DATA_BLOCK "DB_DigIn_I3.6"   // DB138
{ S7_Optimized_Access := 'TRUE' }
VERSION : 0.1
// stored: InstanceOfName FB_DigIn
"FB_DigIn"
BEGIN
END_DATA_BLOCK

DATA_BLOCK "DB_DigIn_I3.7"   // DB139
{ S7_Optimized_Access := 'TRUE' }
VERSION : 0.1
// stored: InstanceOfName FB_DigIn
"FB_DigIn"
BEGIN
END_DATA_BLOCK

DATA_BLOCK "DB_DigIn_I4.0"   // DB140
{ S7_Optimized_Access := 'TRUE' }
VERSION : 0.1
// stored: InstanceOfName FB_DigIn
"FB_DigIn"
BEGIN
END_DATA_BLOCK

DATA_BLOCK "DB_DigIn_I4.1"   // DB141
{ S7_Optimized_Access := 'TRUE' }
VERSION : 0.1
// stored: InstanceOfName FB_DigIn
"FB_DigIn"
BEGIN
END_DATA_BLOCK

DATA_BLOCK "DB_DigIn_I4.2"   // DB142
{ S7_Optimized_Access := 'TRUE' }
VERSION : 0.1
// stored: InstanceOfName FB_DigIn
"FB_DigIn"
BEGIN
END_DATA_BLOCK

DATA_BLOCK "DB_DigIn_I4.3"   // DB143
{ S7_Optimized_Access := 'TRUE' }
VERSION : 0.1
// stored: InstanceOfName FB_DigIn
"FB_DigIn"
BEGIN
END_DATA_BLOCK

DATA_BLOCK "DB_DigIn_I4.4"   // DB144
{ S7_Optimized_Access := 'TRUE' }
VERSION : 0.1
// stored: InstanceOfName FB_DigIn
"FB_DigIn"
BEGIN
END_DATA_BLOCK

DATA_BLOCK "DB_DigIn_I4.5"   // DB145
{ S7_Optimized_Access := 'TRUE' }
VERSION : 0.1
// stored: InstanceOfName FB_DigIn
"FB_DigIn"
BEGIN
END_DATA_BLOCK

DATA_BLOCK "DB_DigIn_I4.6"   // DB146
{ S7_Optimized_Access := 'TRUE' }
VERSION : 0.1
// stored: InstanceOfName FB_DigIn
"FB_DigIn"
BEGIN
END_DATA_BLOCK

DATA_BLOCK "DB_DigIn_I4.7"   // DB147
{ S7_Optimized_Access := 'TRUE' }
VERSION : 0.1
// stored: InstanceOfName FB_DigIn
"FB_DigIn"
BEGIN
END_DATA_BLOCK

DATA_BLOCK "DB_DigIn_I5.0"   // DB148
{ S7_Optimized_Access := 'TRUE' }
VERSION : 0.1
// stored: InstanceOfName FB_DigIn
"FB_DigIn"
BEGIN
END_DATA_BLOCK

DATA_BLOCK "DB_DigIn_I5.1"   // DB149
{ S7_Optimized_Access := 'TRUE' }
VERSION : 0.1
// stored: InstanceOfName FB_DigIn
"FB_DigIn"
BEGIN
END_DATA_BLOCK

DATA_BLOCK "DB_DigIn_I5.2"   // DB150
{ S7_Optimized_Access := 'TRUE' }
VERSION : 0.1
// stored: InstanceOfName FB_DigIn
"FB_DigIn"
BEGIN
END_DATA_BLOCK

DATA_BLOCK "DB_DigIn_I5.3"   // DB151
{ S7_Optimized_Access := 'TRUE' }
VERSION : 0.1
// stored: InstanceOfName FB_DigIn
"FB_DigIn"
BEGIN
END_DATA_BLOCK

DATA_BLOCK "DB_DigIn_I5.4"   // DB152
{ S7_Optimized_Access := 'TRUE' }
VERSION : 0.1
// stored: InstanceOfName FB_DigIn
"FB_DigIn"
BEGIN
END_DATA_BLOCK

DATA_BLOCK "DB_DigIn_I5.5"   // DB153
{ S7_Optimized_Access := 'TRUE' }
VERSION : 0.1
// stored: InstanceOfName FB_DigIn
"FB_DigIn"
BEGIN
END_DATA_BLOCK

DATA_BLOCK "DB_DigIn_I5.6"   // DB154
{ S7_Optimized_Access := 'TRUE' }
VERSION : 0.1
// stored: InstanceOfName FB_DigIn
"FB_DigIn"
BEGIN
END_DATA_BLOCK

DATA_BLOCK "DB_DigIn_I5.7"   // DB155
{ S7_Optimized_Access := 'TRUE' }
VERSION : 0.1
// stored: InstanceOfName FB_DigIn
"FB_DigIn"
BEGIN
END_DATA_BLOCK

DATA_BLOCK "DB_DigIn_I6.0"   // DB156
{ S7_Optimized_Access := 'TRUE' }
VERSION : 0.1
// stored: InstanceOfName FB_DigIn
"FB_DigIn"
BEGIN
END_DATA_BLOCK

DATA_BLOCK "DB_DigIn_I6.1"   // DB157
{ S7_Optimized_Access := 'TRUE' }
VERSION : 0.1
// stored: InstanceOfName FB_DigIn
"FB_DigIn"
BEGIN
END_DATA_BLOCK

DATA_BLOCK "DB_DigIn_I6.2"   // DB158
{ S7_Optimized_Access := 'TRUE' }
VERSION : 0.1
// stored: InstanceOfName FB_DigIn
"FB_DigIn"
BEGIN
END_DATA_BLOCK

DATA_BLOCK "DB_DigIn_I6.3"   // DB159
{ S7_Optimized_Access := 'TRUE' }
VERSION : 0.1
// stored: InstanceOfName FB_DigIn
"FB_DigIn"
BEGIN
END_DATA_BLOCK

DATA_BLOCK "DB_DigIn_I6.4"   // DB160
{ S7_Optimized_Access := 'TRUE' }
VERSION : 0.1
// stored: InstanceOfName FB_DigIn
"FB_DigIn"
BEGIN
END_DATA_BLOCK

DATA_BLOCK "DB_DigIn_I6.5"   // DB161
{ S7_Optimized_Access := 'TRUE' }
VERSION : 0.1
// stored: InstanceOfName FB_DigIn
"FB_DigIn"
BEGIN
END_DATA_BLOCK

DATA_BLOCK "DB_DigIn_I6.6"   // DB162
{ S7_Optimized_Access := 'TRUE' }
VERSION : 0.1
// stored: InstanceOfName FB_DigIn
"FB_DigIn"
BEGIN
END_DATA_BLOCK

DATA_BLOCK "DB_DigIn_I6.7"   // DB163
{ S7_Optimized_Access := 'TRUE' }
VERSION : 0.1
// stored: InstanceOfName FB_DigIn
"FB_DigIn"
BEGIN
END_DATA_BLOCK

DATA_BLOCK "DB_DigIn_I7.0"   // DB164
{ S7_Optimized_Access := 'TRUE' }
VERSION : 0.1
// stored: InstanceOfName FB_DigIn
"FB_DigIn"
BEGIN
END_DATA_BLOCK

DATA_BLOCK "DB_DigIn_I7.1"   // DB165
{ S7_Optimized_Access := 'TRUE' }
VERSION : 0.1
// stored: InstanceOfName FB_DigIn
"FB_DigIn"
BEGIN
END_DATA_BLOCK

DATA_BLOCK "DB_DigIn_I7.2"   // DB166
{ S7_Optimized_Access := 'TRUE' }
VERSION : 0.1
// stored: InstanceOfName FB_DigIn
"FB_DigIn"
BEGIN
END_DATA_BLOCK

DATA_BLOCK "DB_DigIn_I7.3"   // DB167
{ S7_Optimized_Access := 'TRUE' }
VERSION : 0.1
// stored: InstanceOfName FB_DigIn
"FB_DigIn"
BEGIN
END_DATA_BLOCK

DATA_BLOCK "DB_DigIn_I7.4"   // DB168
{ S7_Optimized_Access := 'TRUE' }
VERSION : 0.1
// stored: InstanceOfName FB_DigIn
"FB_DigIn"
BEGIN
END_DATA_BLOCK

DATA_BLOCK "DB_DigIn_I7.5"   // DB169
{ S7_Optimized_Access := 'TRUE' }
VERSION : 0.1
// stored: InstanceOfName FB_DigIn
"FB_DigIn"
BEGIN
END_DATA_BLOCK

DATA_BLOCK "DB_DigIn_I7.6"   // DB170
{ S7_Optimized_Access := 'TRUE' }
VERSION : 0.1
// stored: InstanceOfName FB_DigIn
"FB_DigIn"
BEGIN
END_DATA_BLOCK

DATA_BLOCK "DB_DigIn_I7.7"   // DB171
{ S7_Optimized_Access := 'TRUE' }
VERSION : 0.1
// stored: InstanceOfName FB_DigIn
"FB_DigIn"
BEGIN
END_DATA_BLOCK

DATA_BLOCK "DB_DigOut_Q0.0"   // DB172
{ S7_Optimized_Access := 'TRUE' }
VERSION : 0.1
// stored: InstanceOfName FB_DigOut
"FB_DigOut"
BEGIN
END_DATA_BLOCK

DATA_BLOCK "DB_DigOut_Q0.1"   // DB173
{ S7_Optimized_Access := 'TRUE' }
VERSION : 0.1
// stored: InstanceOfName FB_DigOut
"FB_DigOut"
BEGIN
END_DATA_BLOCK

DATA_BLOCK "DB_DigOut_Q0.2"   // DB174
{ S7_Optimized_Access := 'TRUE' }
VERSION : 0.1
// stored: InstanceOfName FB_DigOut
"FB_DigOut"
BEGIN
END_DATA_BLOCK

DATA_BLOCK "DB_DigOut_Q0.3"   // DB175
{ S7_Optimized_Access := 'TRUE' }
VERSION : 0.1
// stored: InstanceOfName FB_DigOut
"FB_DigOut"
BEGIN
END_DATA_BLOCK

DATA_BLOCK "DB_DigOut_Q0.4"   // DB176
{ S7_Optimized_Access := 'TRUE' }
VERSION : 0.1
// stored: InstanceOfName FB_DigOut
"FB_DigOut"
BEGIN
END_DATA_BLOCK

DATA_BLOCK "DB_DigOut_Q0.5"   // DB177
{ S7_Optimized_Access := 'TRUE' }
VERSION : 0.1
// stored: InstanceOfName FB_DigOut
"FB_DigOut"
BEGIN
END_DATA_BLOCK

DATA_BLOCK "DB_DigOut_Q0.6"   // DB178
{ S7_Optimized_Access := 'TRUE' }
VERSION : 0.1
// stored: InstanceOfName FB_DigOut
"FB_DigOut"
BEGIN
END_DATA_BLOCK

DATA_BLOCK "DB_DigOut_Q0.7"   // DB179
{ S7_Optimized_Access := 'TRUE' }
VERSION : 0.1
// stored: InstanceOfName FB_DigOut
"FB_DigOut"
BEGIN
END_DATA_BLOCK

DATA_BLOCK "DB_DigOut_Q1.0"   // DB180
{ S7_Optimized_Access := 'TRUE' }
VERSION : 0.1
// stored: InstanceOfName FB_DigOut
"FB_DigOut"
BEGIN
END_DATA_BLOCK

DATA_BLOCK "DB_DigOut_Q1.1"   // DB181
{ S7_Optimized_Access := 'TRUE' }
VERSION : 0.1
// stored: InstanceOfName FB_DigOut
"FB_DigOut"
BEGIN
END_DATA_BLOCK

DATA_BLOCK "DB_DigOut_Q1.2"   // DB182
{ S7_Optimized_Access := 'TRUE' }
VERSION : 0.1
// stored: InstanceOfName FB_DigOut
"FB_DigOut"
BEGIN
END_DATA_BLOCK

DATA_BLOCK "DB_DigOut_Q1.3"   // DB183
{ S7_Optimized_Access := 'TRUE' }
VERSION : 0.1
// stored: InstanceOfName FB_DigOut
"FB_DigOut"
BEGIN
END_DATA_BLOCK

DATA_BLOCK "DB_DigOut_Q1.4"   // DB184
{ S7_Optimized_Access := 'TRUE' }
VERSION : 0.1
// stored: InstanceOfName FB_DigOut
"FB_DigOut"
BEGIN
END_DATA_BLOCK

DATA_BLOCK "DB_DigOut_Q1.5"   // DB185
{ S7_Optimized_Access := 'TRUE' }
VERSION : 0.1
// stored: InstanceOfName FB_DigOut
"FB_DigOut"
BEGIN
END_DATA_BLOCK

DATA_BLOCK "DB_DigOut_Q1.6"   // DB186
{ S7_Optimized_Access := 'TRUE' }
VERSION : 0.1
// stored: InstanceOfName FB_DigOut
"FB_DigOut"
BEGIN
END_DATA_BLOCK

DATA_BLOCK "DB_DigOut_Q1.7"   // DB187
{ S7_Optimized_Access := 'TRUE' }
VERSION : 0.1
// stored: InstanceOfName FB_DigOut
"FB_DigOut"
BEGIN
END_DATA_BLOCK

// folder: 2000_Tools

DATA_BLOCK "FB_Bell_DB"   // DB2003
{ S7_Optimized_Access := 'TRUE' }
VERSION : 0.1
// stored: InstanceOfName FB_Bell
"FB_Bell"
BEGIN
END_DATA_BLOCK

// folder: 20_PSM/PSM_DB

DATA_BLOCK "DB_PSM_LC"   // DB20
{ S7_Optimized_Access := 'TRUE' }
VERSION : 0.1
// stored: InstanceOfName FB_PSM_LC
"FB_PSM_LC"
BEGIN
END_DATA_BLOCK

DATA_BLOCK "DB_PSM_Messages"   // DB21
{ S7_Optimized_Access := 'TRUE' }
VERSION : 0.1
// stored: InstanceOfName FB_PSM_Messages
"FB_PSM_Messages"
BEGIN
END_DATA_BLOCK

DATA_BLOCK "DB_PSM_Alarms"   // DB22
{ S7_Optimized_Access := 'TRUE' }
VERSION : 0.1
// stored: InstanceOfName FB_PSM_Alarms
"FB_PSM_Alarms"
BEGIN
END_DATA_BLOCK

// folder: 300_1UZ1_Lifting(LM)/LM_DB

DATA_BLOCK "DB_Lifting_Control"   // DB300
{ S7_Optimized_Access := 'TRUE' }
VERSION : 0.1
// stored: InstanceOfName FB_Lifting_Control
"FB_Lifting_Control"
BEGIN
END_DATA_BLOCK

DATA_BLOCK "DB_LiftUp_Messages"   // DB321
{ S7_Optimized_Access := 'TRUE' }
VERSION : 0.1
// stored: InstanceOfName FB_LiftUp_Messages
"FB_LiftUp_Messages"
BEGIN
END_DATA_BLOCK

// folder: 400_3UZ1_Trolley_movement(TM)/TM_DB

DATA_BLOCK "DB_Trolley_Control"   // DB400
{ S7_Optimized_Access := 'TRUE' }
VERSION : 0.1
// stored: InstanceOfName FB_Trolley_Control
"FB_Trolley_Control"
BEGIN
END_DATA_BLOCK

DATA_BLOCK "DB_Trolley_Messages"   // DB421
{ S7_Optimized_Access := 'TRUE' }
VERSION : 0.1
// stored: InstanceOfName FB_Trolley_Messages
"FB_Trolley_Messages"
BEGIN
END_DATA_BLOCK

// folder: 500_4UZ1_4UZ2_Crane_movement(CM)/CM_DB

DATA_BLOCK "DB_Crane_Control"   // DB500
{ S7_Optimized_Access := 'TRUE' }
VERSION : 0.1
// stored: InstanceOfName FB_Crane_Control
"FB_Crane_Control"
BEGIN
END_DATA_BLOCK

DATA_BLOCK "DB_Crane_Messages"   // DB521
{ S7_Optimized_Access := 'TRUE' }
VERSION : 0.1
// stored: InstanceOfName FB_Crane_Messages
"FB_Crane_Messages"
BEGIN
END_DATA_BLOCK

// folder: 50_Drives/Drives_DB

DATA_BLOCK "DB_CU_U1"   // DB50
{ S7_Optimized_Access := 'TRUE' }
VERSION : 0.1
// stored: InstanceOfName FB_S120_Tel390_CU
"FB_S120_Tel390_CU"
BEGIN
END_DATA_BLOCK

DATA_BLOCK "DB_Drive_1UZ1"   // DB51
{ S7_Optimized_Access := 'TRUE' }
VERSION : 0.1
// stored: InstanceOfName FB_S120_Tel220
"FB_S120_Tel220"
BEGIN
END_DATA_BLOCK

DATA_BLOCK "DB_Drive_3UZ1"   // DB52
{ S7_Optimized_Access := 'TRUE' }
VERSION : 0.1
// stored: InstanceOfName FB_S120_Tel220
"FB_S120_Tel220"
BEGIN
END_DATA_BLOCK

DATA_BLOCK "DB_Drive_4UZ1"   // DB53
{ S7_Optimized_Access := 'TRUE' }
VERSION : 0.1
// stored: InstanceOfName FB_S120_Tel220
"FB_S120_Tel220"
BEGIN
END_DATA_BLOCK

DATA_BLOCK "DB_Drive_4UZ2"   // DB54
{ S7_Optimized_Access := 'TRUE' }
VERSION : 0.1
// stored: InstanceOfName FB_S120_Tel220
"FB_S120_Tel220"
BEGIN
END_DATA_BLOCK

DATA_BLOCK "DB_Drives_Test"   // DB55
{ S7_Optimized_Access := 'TRUE' }
VERSION : 0.1
   VAR
      Sim_On : Bool := False;
      Sim_Reset : Bool := False;
      U1 : Struct   // Блок керування CU320-2PN
         Enable : Bool := True;
         Ack : Bool := False;
      END_STRUCT;
      "1UZ1" : Struct   // Привід підйому
         Enable : Bool := False;
         Ack : Bool := False;
         SpeedSp : Real := 0.0;
         QuickStop : Bool := False;
         CoastStop : Bool := False;
         SimFault : Bool := False;
         SimWarning : Bool := False;
      END_STRUCT;
      "3UZ1" : Struct   // Привод візка
         Enable : Bool := False;
         Ack : Bool := False;
         SpeedSp : Real := 0.0;
         QuickStop : Bool := False;
         CoastStop : Bool := False;
         SimFault : Bool := False;
         SimWarning : Bool := False;
      END_STRUCT;
      "4UZ1" : Struct   // Привод моста 1
         Enable : Bool := False;
         Ack : Bool := False;
         SpeedSp : Real := 0.0;
         QuickStop : Bool := False;
         CoastStop : Bool := False;
         SimFault : Bool := False;
         SimWarning : Bool := False;
      END_STRUCT;
      "4UZ2" : Struct   // Привод моста 2
         Enable : Bool := False;
         Ack : Bool := False;
         SpeedSp : Real := 0.0;
         QuickStop : Bool := False;
         CoastStop : Bool := False;
         SimFault : Bool := False;
         SimWarning : Bool := False;
      END_STRUCT;
   END_VAR
BEGIN
END_DATA_BLOCK

// folder: 600_Diagnostic

DATA_BLOCK "FB_DIAG_SCALANCE_NODE_DB"   // DB609
{ S7_Optimized_Access := 'TRUE' }
AUTHOR : PIA
FAMILY : System
VERSION : 0.1
// stored: InstanceOfName FB_DIAG_NODE
"FB_DIAG_NODE"
BEGIN
END_DATA_BLOCK

DATA_BLOCK "DB_HMI_Connection"   // DB631
{ S7_Optimized_Access := 'FALSE' }
VERSION : 0.1
// DB631. Постійна ознака доступності даних ПЛК для HMI. Не потребує виклику в OB1. Опитування RUN/STOP використовує існуючу область HMI_DB.wCoordination.
   VAR
      Available : Bool := true;   // Постійне TRUE для перевірки звʼязку з HMI. Після помилки звʼязку панель локально підставляє FALSE; значення у DB не змінюється.
   END_VAR
BEGIN
END_DATA_BLOCK

// folder: 600_Diagnostic/Diag_DB

DATA_BLOCK "DB_SCALANCE"   // DB600
{ S7_Optimized_Access := 'TRUE' }
AUTHOR : PIA
FAMILY : System
VERSION : 0.1
// stored: InstanceOfName FB_DIAG_SCALANCE
"FB_DIAG_SCALANCE"
BEGIN
END_DATA_BLOCK

DATA_BLOCK "DB_DIAG_NODE"   // DB601
{ S7_Optimized_Access := 'TRUE' }
AUTHOR : PIA
FAMILY : System
VERSION : 0.1
// stored: InstanceOfName FB_DIAG_NODE
"FB_DIAG_NODE"
BEGIN
END_DATA_BLOCK

DATA_BLOCK "DB_DIAG_ENC_1BR_NODE"   // DB602
{ S7_Optimized_Access := 'TRUE' }
AUTHOR : PIA
FAMILY : System
VERSION : 0.1
// stored: InstanceOfName FB_DIAG_NODE
"FB_DIAG_NODE"
BEGIN
END_DATA_BLOCK

DATA_BLOCK "DB_DIAG_ENC_3BR_NODE"   // DB603
{ S7_Optimized_Access := 'TRUE' }
AUTHOR : PIA
FAMILY : System
VERSION : 0.1
// stored: InstanceOfName FB_DIAG_NODE
"FB_DIAG_NODE"
BEGIN
END_DATA_BLOCK

DATA_BLOCK "DB_DIAG_ENC_4BR1_NODE"   // DB604
{ S7_Optimized_Access := 'TRUE' }
AUTHOR : PIA
FAMILY : System
VERSION : 0.1
// stored: InstanceOfName FB_DIAG_NODE
"FB_DIAG_NODE"
BEGIN
END_DATA_BLOCK

DATA_BLOCK "DB_DIAG_ENC_4BR2_NODE"   // DB605
{ S7_Optimized_Access := 'TRUE' }
AUTHOR : PIA
FAMILY : System
VERSION : 0.1
// stored: InstanceOfName FB_DIAG_NODE
"FB_DIAG_NODE"
BEGIN
END_DATA_BLOCK

DATA_BLOCK "DB_DIAG_CU320_NODE"   // DB606
{ S7_Optimized_Access := 'TRUE' }
AUTHOR : PIA
FAMILY : System
VERSION : 0.1
// stored: InstanceOfName FB_DIAG_NODE
"FB_DIAG_NODE"
BEGIN
END_DATA_BLOCK

DATA_BLOCK "DB_DIAG_SCALANCE"   // DB607
{ S7_Optimized_Access := 'TRUE' }
AUTHOR : PIA
FAMILY : System
VERSION : 0.1
// stored: InstanceOfName FB_DIAG_SCALANCE
"FB_DIAG_SCALANCE"
BEGIN
END_DATA_BLOCK

DATA_BLOCK "DB_Diagnostics_Messages"   // DB621
{ S7_Optimized_Access := 'TRUE' }
VERSION : 0.1
// stored: InstanceOfName FB_Diagnostics_Messages
"FB_Diagnostics_Messages"
BEGIN
END_DATA_BLOCK

DATA_BLOCK "DB_Diag_Prof"   // DB630
{ S7_Optimized_Access := 'TRUE' }
VERSION : 0.1
// stored: InstanceOfName FB_Diag_MRP
"FB_Diag_MRP"
BEGIN
END_DATA_BLOCK

// folder: 700_Calibration

DATA_BLOCK "DB_Calibration"   // DB700
{ S7_Optimized_Access := 'TRUE' }
VERSION : 0.1
   VAR
      Hoist : Struct   // Підйом
         Start : Bool := FALSE;   // Запуск процедури калібровки
         Reset : Bool := FALSE;   // Скидання сіквенсера та статусу калібровки
         ResetDiagMem : Bool := FALSE;   // Скидання діагностики - пам'ять фронту
         Abort : Bool := FALSE;   // Ручне переривання процедури
         ForceCalibrated : Bool := FALSE;   // Примусове встановлення статусу калібровки для ПНР
         PresetValueRaw : DInt := DINT#130250000;   // Значення preset для точки калібровки, інкременти
         TimeoutA : Time := T#1m;   // Максимальний час очікування початку руху
         TimeoutB : Time := T#5m;   // Максимальний час виконання пошуку реперної точки
         StandstillSpeed_rpm : Real := 5.0;   // Максимальна швидкість для визначення зупинки ПЧ
         StandstillConfirm : Time := T#500ms;   // Час підтвердження стану повної зупинки
         ReferencePosition_mm : LReal := 23500.0;   // Жорстко задана координата реперної точки 1K1, мм.
         VirtualOffset_mm : LReal := 0.0;   // Віртуальне зміщення координати реперної точки, визначається під час ПНР.
         TravelAfterReference_mm : LReal := 0.0;   // Шлях, пройдений механізмом після спадного фронту 1K1 до повної зупинки, мм.
         PresetTargetPosition_mm : LReal := 0.0;   // Цільова координата механізму в момент preset з урахуванням реперної точки, virtual offset та шляху після репера.
         PresetValueRawValid : Bool := FALSE;   // TRUE — розраховане raw-значення може бути використане для preset енкодера.
         PresetCalculationValid : Bool := FALSE;   // TRUE — зворотний розрахунок mm → raw успішно виконаний.
         PresetConfigurationValid : Bool := FALSE;   // TRUE — контрольні точки масштабування та допустимий raw-діапазон задані коректно.
         PresetInConfiguredRange : Bool := FALSE;   // TRUE — цільова координата preset знаходиться в налаштованому діапазоні масштабування.
         PresetInRawRange : Bool := FALSE;   // TRUE — розраховане raw-значення знаходиться в допустимому діапазоні енкодера.
         PresetScale_mm_per_count : LReal := 0.0;   // Розрахований коефіцієнт масштабування, мм на один raw-count.
         PresetCalculatedRaw : LReal := 0.0;   // Розраховане raw-значення до перетворення в DINT. Використовується для діагностики та ПНР.
         PresetCalcStatus : Word := W#16#0000;   // Діагностичне слово функції FC_PositionToRaw.
      END_STRUCT;
      Trolley : Struct   // Візок
         Start : Bool := FALSE;   // Запуск процедури калібровки
         Reset : Bool := FALSE;   // Скидання сіквенсера та статусу калібровки
         ResetDiagMem : Bool := FALSE;   // Скидання діагностики - пам'ять фронту
         Abort : Bool := FALSE;   // Ручне переривання процедури
         ForceCalibrated : Bool := FALSE;   // Примусове встановлення статусу калібровки для ПНР
         PresetValueRaw : DInt := DINT#119305476;   // Значення preset для точки калібровки, інкременти
         TimeoutA : Time := T#1m;   // Максимальний час очікування початку руху
         TimeoutB : Time := T#5m;   // Максимальний час виконання пошуку реперної точки
         StandstillSpeed_rpm : Real := 5.0;   // Максимальна швидкість для визначення зупинки ПЧ
         StandstillConfirm : Time := T#500ms;   // Час підтвердження стану повної зупинки
         HoistPositionMin_mm : LReal := 23750.0;   // Нижня межа допустимої позиції підйому
         HoistPositionMax_mm : LReal := 23900.0;   // Верхня межа допустимої позиції підйому
         ReferencePosition_mm : LReal := 7775.0;   // Жорстко задана координата реперної точки 3K1, мм.
         VirtualOffset_mm : LReal := 0.0;   // Віртуальне зміщення координати реперної точки, визначається під час ПНР.
         TravelAfterReference_mm : LReal := 0.0;   // Шлях, пройдений механізмом після спадного фронту 3K1 до повної зупинки, мм.
         PresetTargetPosition_mm : LReal := 0.0;   // Цільова координата механізму в момент preset з урахуванням реперної точки, virtual offset та шляху після репера.
         PresetValueRawValid : Bool := FALSE;   // TRUE — розраховане raw-значення може бути використане для preset енкодера.
         PresetCalculationValid : Bool := FALSE;   // TRUE — зворотний розрахунок mm → raw успішно виконаний.
         PresetConfigurationValid : Bool := FALSE;   // TRUE — контрольні точки масштабування та допустимий raw-діапазон задані коректно.
         PresetInConfiguredRange : Bool := FALSE;   // TRUE — цільова координата preset знаходиться в налаштованому діапазоні масштабування.
         PresetInRawRange : Bool := FALSE;   // TRUE — розраховане raw-значення знаходиться в допустимому діапазоні енкодера.
         PresetScale_mm_per_count : LReal := 0.0;   // Розрахований коефіцієнт масштабування, мм на один raw-count.
         PresetCalculatedRaw : LReal := 0.0;   // Розраховане raw-значення до перетворення в DINT. Використовується для діагностики та ПНР.
         PresetCalcStatus : Word := W#16#0000;   // Діагностичне слово функції FC_PositionToRaw.
      END_STRUCT;
      Crane : Struct   // Кран
         Start : Bool := FALSE;   // Запуск процедури калібровки
         Reset : Bool := FALSE;   // Скидання сіквенсера та статусу калібровки
         ResetDiagMem : Bool := FALSE;   // Скидання діагностики - пам'ять фронту
         Abort : Bool := FALSE;   // Ручне переривання процедури
         ForceCalibrated : Bool := FALSE;   // Примусове встановлення статусу калібровки для ПНР
         PresetValueRaw1 : DInt := DINT#11061828;   // Значення preset для точки калібровки, інкременти
         PresetValueRaw2 : DInt := DINT#11061828;   // Значення preset для точки калібровки, інкременти
         TimeoutA : Time := T#1m;   // Максимальний час очікування початку руху
         TimeoutB : Time := T#5m;   // Максимальний час виконання пошуку реперної точки
         StandstillSpeed_rpm : Real := 5.0;   // Максимальна швидкість для визначення зупинки ПЧ
         StandstillConfirm : Time := T#500ms;   // Час підтвердження стану повної зупинки
         HoistPositionMin_mm : LReal := 23750.0;   // Нижня межа допустимої позиції підйому
         HoistPositionMax_mm : LReal := 23900.0;   // Верхня межа допустимої позиції підйому
         PresetServiceEnable : Bool := FALSE;   // Загальний дозвіл сервісного preset 4BR1/4BR2
         PresetPermit : Bool := FALSE;   // Загальний дозвіл виконання preset 4BR1/4BR2
         PresetStart : Bool := FALSE;   // Загальний імпульс запуску preset 4BR1/4BR2
         MaxEncoderDifference_mm : LReal := 50.0;   // Максимальна розбіжність 4BR1 та 4BR2
         ReferencePosition_mm : LReal := 900.0;   // Жорстко задана координата реперної точки 4K1, мм.
         VirtualOffset_mm : LReal := 0.0;   // Віртуальне зміщення координати реперної точки, визначається під час ПНР.
         TravelAfterReference1_mm : LReal := 0.0;   // Шлях, пройдений механізмом після спадного фронту 4K1 до повної зупинки, мм.
         TravelAfterReference2_mm : LReal := 0.0;   // Шлях, пройдений механізмом після спадного фронту 4K1 до повної зупинки, мм.
         PresetTargetPosition1_mm : LReal := 0.0;   // Цільова координата механізму в момент preset з урахуванням реперної точки, virtual offset та шляху після репера.
         PresetTargetPosition2_mm : LReal := 0.0;   // Цільова координата механізму в момент preset з урахуванням реперної точки, virtual offset та шляху після репера.
         PresetValueRaw1Valid : Bool := FALSE;   // TRUE — розраховане raw-значення може бути використане для preset енкодера.
         PresetValueRaw2Valid : Bool := FALSE;   // TRUE — розраховане raw-значення може бути використане для preset енкодера.
         PresetCalculation1Valid : Bool := FALSE;   // TRUE — зворотний розрахунок mm → raw успішно виконаний.
         PresetCalculation2Valid : Bool := FALSE;   // TRUE — зворотний розрахунок mm → raw успішно виконаний.
         PresetConfiguration1Valid : Bool := FALSE;   // TRUE — контрольні точки масштабування та допустимий raw-діапазон задані коректно.
         PresetConfiguration2Valid : Bool := FALSE;   // TRUE — контрольні точки масштабування та допустимий raw-діапазон задані коректно.
         Preset1InConfiguredRange : Bool := FALSE;   // TRUE — цільова координата preset знаходиться в налаштованому діапазоні масштабування.
         Preset2InConfiguredRange : Bool := FALSE;   // TRUE — цільова координата preset знаходиться в налаштованому діапазоні масштабування.
         Preset1InRawRange : Bool := FALSE;   // TRUE — розраховане raw-значення знаходиться в допустимому діапазоні енкодера.
         Preset2InRawRange : Bool := FALSE;   // TRUE — розраховане raw-значення знаходиться в допустимому діапазоні енкодера.
         PresetScale1_mm_per_count : LReal := 0.0;   // Розрахований коефіцієнт масштабування, мм на один raw-count.
         PresetScale2_mm_per_count : LReal := 0.0;   // Розрахований коефіцієнт масштабування, мм на один raw-count.
         PresetCalculatedRaw1 : LReal := 0.0;   // Розраховане raw-значення до перетворення в DINT. Використовується для діагностики та ПНР.
         PresetCalculatedRaw2 : LReal := 0.0;   // Розраховане raw-значення до перетворення в DINT. Використовується для діагностики та ПНР.
         PresetCalcStatus1 : Word := W#16#0000;   // Діагностичне слово функції FC_PositionToRaw.
         PresetCalcStatus2 : Word := W#16#0000;   // Діагностичне слово функції FC_PositionToRaw.
      END_STRUCT;
   END_VAR
BEGIN
END_DATA_BLOCK

// folder: 700_Calibration/Crane

DATA_BLOCK "DB_CraneCalibration"   // DB703
{ S7_Optimized_Access := 'TRUE' }
VERSION : 0.1
// stored: InstanceOfName FB_CraneCalibration
"FB_CraneCalibration"
BEGIN
END_DATA_BLOCK

DATA_BLOCK "DB_CraneCalibrationDiag"   // DB713
{ S7_Optimized_Access := 'TRUE' }
VERSION : 0.1
// stored: InstanceOfName FB_CraneCalibrationDiag
"FB_CraneCalibrationDiag"
BEGIN
END_DATA_BLOCK

// folder: 700_Calibration/Hoist/Lifting

DATA_BLOCK "DB_HoistCalibration"   // DB701
{ S7_Optimized_Access := 'TRUE' }
VERSION : 0.1
// stored: InstanceOfName FB_HoistCalibration
"FB_HoistCalibration"
BEGIN
END_DATA_BLOCK

DATA_BLOCK "DB_HoistCalibrationDiag"   // DB711
{ S7_Optimized_Access := 'TRUE' }
VERSION : 0.1
// stored: InstanceOfName FB_HoistCalibrationDiag
"FB_HoistCalibrationDiag"
BEGIN
END_DATA_BLOCK

// folder: 700_Calibration/Trolley

DATA_BLOCK "DB_TrolleyCalibration"   // DB702
{ S7_Optimized_Access := 'TRUE' }
VERSION : 0.1
// stored: InstanceOfName FB_TrolleyCalibration
"FB_TrolleyCalibration"
BEGIN
END_DATA_BLOCK

DATA_BLOCK "DB_TrolleyCalibrationDiag"   // DB712
{ S7_Optimized_Access := 'TRUE' }
VERSION : 0.1
// stored: InstanceOfName FB_TrolleyCalibrationDiag
"FB_TrolleyCalibrationDiag"
BEGIN
END_DATA_BLOCK

// folder: 70_FireAlarm

DATA_BLOCK "DB_FireAlarm"   // DB70
{ S7_Optimized_Access := 'TRUE' }
VERSION : 0.1
// stored: InstanceOfName FB_FireAlarm
"FB_FireAlarm"
BEGIN
END_DATA_BLOCK

// folder: 80_Encoders/Encoders_DB

DATA_BLOCK "DB_EncCom_1BR"   // DB80
{ S7_Optimized_Access := 'TRUE' }
VERSION : 0.1
// stored: InstanceOfName FB_Enc_Tlg89_Com
"FB_Enc_Tlg89_Com"
BEGIN
END_DATA_BLOCK

DATA_BLOCK "DB_EncCom_3BR"   // DB81
{ S7_Optimized_Access := 'TRUE' }
VERSION : 0.1
// stored: InstanceOfName FB_Enc_Tlg89_Com
"FB_Enc_Tlg89_Com"
BEGIN
END_DATA_BLOCK

DATA_BLOCK "DB_EncCom_4BR1"   // DB82
{ S7_Optimized_Access := 'TRUE' }
VERSION : 0.1
// stored: InstanceOfName FB_Enc_Tlg89_Com
"FB_Enc_Tlg89_Com"
BEGIN
END_DATA_BLOCK

DATA_BLOCK "DB_EncCom_4BR2"   // DB83
{ S7_Optimized_Access := 'TRUE' }
VERSION : 0.1
// stored: InstanceOfName FB_Enc_Tlg89_Com
"FB_Enc_Tlg89_Com"
BEGIN
END_DATA_BLOCK

DATA_BLOCK "DB_EncCtrl"   // DB84
{ S7_Optimized_Access := 'TRUE' }
VERSION : 0.1
   VAR
      "1BR" : Struct   // Керування енкодером 1BR
         ResetSimulation : Bool := FALSE;   // Імпульсна команда скидання симуляції енкодера. Вмикати коротко TRUE, потім назад FALSE.
         MotionEnable : Bool := FALSE;   // Розрахунковий дозвіл руху симулятора. Формується в OB30 від CmdUp/CmdDown.
         VelocityCommandRawPerSec : LReal := 0.0;   // Розрахункова команда швидкості для FB_Enc_Tlg89_Sim. Формується в OB30.
         QuickStop : Bool := FALSE;   // Команда швидкої зупинки симулятора.
         InjectCommunicationFault : Bool := FALSE;   // Імітація втрати зв’язку з енкодером. Для нормального тесту має бути FALSE.
         InjectControlInactive : Bool := FALSE;   // Імітація відсутності підтвердження керування від енкодера. Для нормального тесту має бути FALSE.
         InjectEncoderFault : Bool := FALSE;   // Імітація активної помилки енкодера. Формує ZSW2_ENC bit 3.
         InjectEncoderAlarm : Bool := FALSE;   // Імітація попередження енкодера. Формує ZSW2_ENC bit 7.
         ForceInvalidPosition : Bool := FALSE;   // Примусово робить положення недостовірним. Скидає ZSW2_ENC bit 1.
         ForceInvalidVelocity : Bool := FALSE;   // Примусово робить швидкість недостовірною. Скидає ZSW2_ENC bit 2.
         FreezeEncoderLife : Bool := FALSE;   // Зупинка encoder sign-of-life. Для нормального тесту має бути FALSE.
         InjectMasterLifeFault : Bool := FALSE;   // Імітація помилки master sign-of-life від PLC.
         TestModeActive : Bool := FALSE;   // Загальний прапор тестового режиму. Використовується для автоматичного керування симуляцією.
         CmdUp : Bool := FALSE;   // Ручна тестова команда руху вгору.
         CmdDown : Bool := FALSE;   // Ручна тестова команда руху вниз.
         SpeedCommandRawPerSec : LReal := 500.0;   // Базова тестова швидкість у raw-count/сек. Для першого тесту залишити 500.0.
         PositiveDirectionIsUp : Bool := TRUE;   // TRUE = позитивний напрям raw-позиції відповідає руху вгору.
         DirectionConflict : Bool := FALSE;   // Ознака одночасної команди CmdUp і CmdDown. Формується в OB30.
         CalibrationEnable : Bool := FALSE;   // Інженерний дозвіл калібровки в FB_HoistPosition.
         CalibrationStart : Bool := FALSE;   // Імпульс запуску калібровки. Вмикати коротко TRUE, потім назад FALSE.
         ResetCalibrationLost : Bool := FALSE;   // Імпульс квітування діагностики втрати калібровки.
         PresetServiceEnable : Bool := FALSE;   // Дозвіл сервісної preset-функції в FB_Enc_Tlg89_Com. Для нормальної роботи має бути FALSE.
         PresetPermit : Bool := FALSE;   // Дозвіл виконання preset від логіки ПЛК. Має бути TRUE тільки коли механізм стоїть і активний сервісний режим.
         PresetStart : Bool := FALSE;   // Імпульс запуску preset через Telegram 89.
         PresetValueRaw : DInt := 0;   // Значення preset у raw-count. Наприклад 50000.
         DriveAtStandstill : Bool;   // Признак зупинки привода
         DriveFrequencyZero : Bool;   // Нульова частота з приводу
      END_STRUCT;
      "3BR" : Struct   // Керування енкодером 3BR
         ResetSimulation : Bool := FALSE;   // Імпульсна команда скидання симуляції енкодера. Вмикати коротко TRUE, потім назад FALSE.
         MotionEnable : Bool := FALSE;   // Розрахунковий дозвіл руху симулятора. Формується в OB30 від CmdUp/CmdDown.
         VelocityCommandRawPerSec : LReal := 0.0;   // Розрахункова команда швидкості для FB_Enc_Tlg89_Sim. Формується в OB30.
         QuickStop : Bool := FALSE;   // Команда швидкої зупинки симулятора.
         InjectCommunicationFault : Bool := FALSE;   // Імітація втрати зв’язку з енкодером. Для нормального тесту має бути FALSE.
         InjectControlInactive : Bool := FALSE;   // Імітація відсутності підтвердження керування від енкодера. Для нормального тесту має бути FALSE.
         InjectEncoderFault : Bool := FALSE;   // Імітація активної помилки енкодера. Формує ZSW2_ENC bit 3.
         InjectEncoderAlarm : Bool := FALSE;   // Імітація попередження енкодера. Формує ZSW2_ENC bit 7.
         ForceInvalidPosition : Bool := FALSE;   // Примусово робить положення недостовірним. Скидає ZSW2_ENC bit 1.
         ForceInvalidVelocity : Bool := FALSE;   // Примусово робить швидкість недостовірною. Скидає ZSW2_ENC bit 2.
         FreezeEncoderLife : Bool := FALSE;   // Зупинка encoder sign-of-life. Для нормального тесту має бути FALSE.
         InjectMasterLifeFault : Bool := FALSE;   // Імітація помилки master sign-of-life від PLC.
         TestModeActive : Bool := TRUE;   // Загальний прапор тестового режиму. Використовується для автоматичного керування симуляцією.
         CmdUp : Bool := FALSE;   // Ручна тестова команда руху вгору.
         CmdDown : Bool := FALSE;   // Ручна тестова команда руху вниз.
         SpeedCommandRawPerSec : LReal := 500.0;   // Базова тестова швидкість у raw-count/сек. Для першого тесту залишити 500.0.
         PositiveDirectionIsUp : Bool := TRUE;   // TRUE = позитивний напрям raw-позиції відповідає руху вгору.
         DirectionConflict : Bool := FALSE;   // Ознака одночасної команди CmdUp і CmdDown. Формується в OB30.
         CalibrationEnable : Bool := FALSE;   // Інженерний дозвіл калібровки в FB_HoistPosition.
         CalibrationStart : Bool := FALSE;   // Імпульс запуску калібровки. Вмикати коротко TRUE, потім назад FALSE.
         ResetCalibrationLost : Bool := FALSE;   // Імпульс квітування діагностики втрати калібровки.
         PresetServiceEnable : Bool := FALSE;   // Дозвіл сервісної preset-функції в FB_Enc_Tlg89_Com. Для нормальної роботи має бути FALSE.
         PresetPermit : Bool := FALSE;   // Дозвіл виконання preset від логіки ПЛК. Має бути TRUE тільки коли механізм стоїть і активний сервісний режим.
         PresetStart : Bool := FALSE;   // Імпульс запуску preset через Telegram 89.
         PresetValueRaw : DInt := 0;   // Значення preset у raw-count. Наприклад 50000.
         DriveAtStandstill : Bool;   // Признак зупинки привода
         DriveFrequencyZero : Bool;   // Нульова частота з приводу
      END_STRUCT;
      "4BR1" : Struct   // Керування енкодером 4BR1
         ResetSimulation : Bool := FALSE;   // Імпульсна команда скидання симуляції енкодера. Вмикати коротко TRUE, потім назад FALSE.
         MotionEnable : Bool := FALSE;   // Розрахунковий дозвіл руху симулятора. Формується в OB30 від CmdUp/CmdDown.
         VelocityCommandRawPerSec : LReal := 0.0;   // Розрахункова команда швидкості для FB_Enc_Tlg89_Sim. Формується в OB30.
         QuickStop : Bool := FALSE;   // Команда швидкої зупинки симулятора.
         InjectCommunicationFault : Bool := FALSE;   // Імітація втрати зв’язку з енкодером. Для нормального тесту має бути FALSE.
         InjectControlInactive : Bool := FALSE;   // Імітація відсутності підтвердження керування від енкодера. Для нормального тесту має бути FALSE.
         InjectEncoderFault : Bool := FALSE;   // Імітація активної помилки енкодера. Формує ZSW2_ENC bit 3.
         InjectEncoderAlarm : Bool := FALSE;   // Імітація попередження енкодера. Формує ZSW2_ENC bit 7.
         ForceInvalidPosition : Bool := FALSE;   // Примусово робить положення недостовірним. Скидає ZSW2_ENC bit 1.
         ForceInvalidVelocity : Bool := FALSE;   // Примусово робить швидкість недостовірною. Скидає ZSW2_ENC bit 2.
         FreezeEncoderLife : Bool := FALSE;   // Зупинка encoder sign-of-life. Для нормального тесту має бути FALSE.
         InjectMasterLifeFault : Bool := FALSE;   // Імітація помилки master sign-of-life від PLC.
         TestModeActive : Bool := TRUE;   // Загальний прапор тестового режиму. Використовується для автоматичного керування симуляцією.
         CmdUp : Bool := FALSE;   // Ручна тестова команда руху вгору.
         CmdDown : Bool := FALSE;   // Ручна тестова команда руху вниз.
         SpeedCommandRawPerSec : LReal := 500.0;   // Базова тестова швидкість у raw-count/сек. Для першого тесту залишити 500.0.
         PositiveDirectionIsUp : Bool := TRUE;   // TRUE = позитивний напрям raw-позиції відповідає руху вгору.
         DirectionConflict : Bool := FALSE;   // Ознака одночасної команди CmdUp і CmdDown. Формується в OB30.
         CalibrationEnable : Bool := FALSE;   // Інженерний дозвіл калібровки в FB_HoistPosition.
         CalibrationStart : Bool := FALSE;   // Імпульс запуску калібровки. Вмикати коротко TRUE, потім назад FALSE.
         ResetCalibrationLost : Bool := FALSE;   // Імпульс квітування діагностики втрати калібровки.
         PresetServiceEnable : Bool := FALSE;   // Дозвіл сервісної preset-функції в FB_Enc_Tlg89_Com. Для нормальної роботи має бути FALSE.
         PresetPermit : Bool := FALSE;   // Дозвіл виконання preset від логіки ПЛК. Має бути TRUE тільки коли механізм стоїть і активний сервісний режим.
         PresetStart : Bool := FALSE;   // Імпульс запуску preset через Telegram 89.
         PresetValueRaw : DInt := 0;   // Значення preset у raw-count. Наприклад 50000.
         DriveAtStandstill : Bool;   // Признак зупинки привода
         DriveFrequencyZero : Bool;   // Нульова частота з приводу
      END_STRUCT;
      "4BR2" : Struct   // Керування енкодером 4BR2
         ResetSimulation : Bool := FALSE;   // Імпульсна команда скидання симуляції енкодера. Вмикати коротко TRUE, потім назад FALSE.
         MotionEnable : Bool := FALSE;   // Розрахунковий дозвіл руху симулятора. Формується в OB30 від CmdUp/CmdDown.
         VelocityCommandRawPerSec : LReal := 0.0;   // Розрахункова команда швидкості для FB_Enc_Tlg89_Sim. Формується в OB30.
         QuickStop : Bool := FALSE;   // Команда швидкої зупинки симулятора.
         InjectCommunicationFault : Bool := FALSE;   // Імітація втрати зв’язку з енкодером. Для нормального тесту має бути FALSE.
         InjectControlInactive : Bool := FALSE;   // Імітація відсутності підтвердження керування від енкодера. Для нормального тесту має бути FALSE.
         InjectEncoderFault : Bool := FALSE;   // Імітація активної помилки енкодера. Формує ZSW2_ENC bit 3.
         InjectEncoderAlarm : Bool := FALSE;   // Імітація попередження енкодера. Формує ZSW2_ENC bit 7.
         ForceInvalidPosition : Bool := FALSE;   // Примусово робить положення недостовірним. Скидає ZSW2_ENC bit 1.
         ForceInvalidVelocity : Bool := FALSE;   // Примусово робить швидкість недостовірною. Скидає ZSW2_ENC bit 2.
         FreezeEncoderLife : Bool := FALSE;   // Зупинка encoder sign-of-life. Для нормального тесту має бути FALSE.
         InjectMasterLifeFault : Bool := FALSE;   // Імітація помилки master sign-of-life від PLC.
         TestModeActive : Bool := TRUE;   // Загальний прапор тестового режиму. Використовується для автоматичного керування симуляцією.
         CmdUp : Bool := FALSE;   // Ручна тестова команда руху вгору.
         CmdDown : Bool := FALSE;   // Ручна тестова команда руху вниз.
         SpeedCommandRawPerSec : LReal := 500.0;   // Базова тестова швидкість у raw-count/сек. Для першого тесту залишити 500.0.
         PositiveDirectionIsUp : Bool := TRUE;   // TRUE = позитивний напрям raw-позиції відповідає руху вгору.
         DirectionConflict : Bool := FALSE;   // Ознака одночасної команди CmdUp і CmdDown. Формується в OB30.
         CalibrationEnable : Bool := FALSE;   // Інженерний дозвіл калібровки в FB_HoistPosition.
         CalibrationStart : Bool := FALSE;   // Імпульс запуску калібровки. Вмикати коротко TRUE, потім назад FALSE.
         ResetCalibrationLost : Bool := FALSE;   // Імпульс квітування діагностики втрати калібровки.
         PresetServiceEnable : Bool := FALSE;   // Дозвіл сервісної preset-функції в FB_Enc_Tlg89_Com. Для нормальної роботи має бути FALSE.
         PresetPermit : Bool := FALSE;   // Дозвіл виконання preset від логіки ПЛК. Має бути TRUE тільки коли механізм стоїть і активний сервісний режим.
         PresetStart : Bool := FALSE;   // Імпульс запуску preset через Telegram 89.
         PresetValueRaw : DInt := 0;   // Значення preset у raw-count. Наприклад 50000.
         DriveAtStandstill : Bool;   // Признак зупинки привода
         DriveFrequencyZero : Bool;   // Нульова частота з приводу
      END_STRUCT;
   END_VAR
BEGIN
END_DATA_BLOCK

DATA_BLOCK "DB_EncoderScaling"   // DB87
{ S7_Optimized_Access := 'TRUE' }
VERSION : 0.1
   VAR
      Enc_1BR : Struct
         RawPoint1 : DInt := 1000000;   // Raw-значення, яке відповідає 0 мм.
         PositionPoint1_mm : LReal := 0.0;   // Перша координата, мм.
         RawPoint2 : DInt := 133_000_000;   // Raw-значення максимальної координати.
         PositionPoint2_mm : LReal := 24000.0;   // Максимальна координата за ТЗ. / Максимальна координата підйому за ТЗ.
         Position_mm : LReal := 16106.0110909091;   // Поточне масштабоване положення.
         PositionRounded_mm : DInt := 16106;   // Положення, округлене до цілого мм.
         PositionValid : Bool := TRUE;   // Положення придатне для штатного використання.
         CalculationValid : Bool := TRUE;   // Розрахунок виконано за достовірним raw.
         ConfigurationValid : Bool := TRUE;   // Контрольні точки задані коректно.
         InConfiguredRange : Bool := TRUE;   // Raw знаходиться між контрольними точками.
         BelowConfiguredRange : Bool := FALSE;   // Raw нижче налаштованого діапазону.
         AboveConfiguredRange : Bool := FALSE;   // Raw вище налаштованого діапазону.
         Scale_mm_per_count : LReal := 0.000181818181818182;   // Розрахований коефіцієнт масштабування.
         Status : Word := 16#0060;   // Діагностичне слово.
         ProgSwitches : Struct   // Програмні вимикачі
            DownEndPosition : Bool := FALSE;   // Досягнута крайня нижня позиція
            DownEmergencyLimit : Bool := FALSE;   // Досягнута позиція аварійного кінцевика при опусканні
            DownEncoderLimit : Bool := FALSE;   // Досягнута програмна межа по енкодеру при опусканні
            DownPreStop : Bool := FALSE;   // Активна зона технологічного передзупину при опусканні
            UpPreStop : Bool := FALSE;   // Активна зона технологічного передзупину при підйомі
            UpEncoderLimit : Bool := FALSE;   // Досягнута програмна межа по енкодеру при підйомі
            UpEmergencyLimit : Bool := FALSE;   // Досягнута позиція аварійного кінцевика при підйомі
            UpEndPosition : Bool := FALSE;   // Досягнута крайня верхня позиція
         END_STRUCT;
      END_STRUCT;
      Enc_3BR : Struct
         RawPoint1 : DInt := 1000000;   // Raw-значення, яке відповідає 0 мм.
         PositionPoint1_mm : LReal := 0.0;   // Перша координата, мм.
         RawPoint2 : DInt := 133_000_000;   // Raw-значення максимальної координати.
         PositionPoint2_mm : LReal := 8675.0;   // Максимальна координата за ТЗ. / Максимальна координата підйому за ТЗ.
         Position_mm : LReal := 7500.00318977273;   // Поточне масштабоване положення.
         PositionRounded_mm : DInt := 7500;   // Положення, округлене до цілого мм.
         PositionValid : Bool := TRUE;   // Положення придатне для штатного використання.
         CalculationValid : Bool := TRUE;   // Розрахунок виконано за достовірним raw.
         ConfigurationValid : Bool := TRUE;   // Контрольні точки задані коректно.
         InConfiguredRange : Bool := TRUE;   // Raw знаходиться між контрольними точками.
         BelowConfiguredRange : Bool := FALSE;   // Raw нижче налаштованого діапазону.
         AboveConfiguredRange : Bool := FALSE;   // Raw вище налаштованого діапазону.
         Scale_mm_per_count : LReal := 6.5719696969697E-05;   // Розрахований коефіцієнт масштабування.
         Status : Word := 16#0060;   // Діагностичне слово.
         ProgSwitches : Struct   // Програмні вимикачі
            BackBuffer : Bool := FALSE;   // TRUE = досягнута або перевищена позиція буфера назад
            BackEmergencyLimit : Bool := FALSE;   // TRUE = досягнута позиція аварійного кінцевика назад
            BackEncoderLimit : Bool := FALSE;   // TRUE = досягнута програмна межа по енкодеру назад
            BackPreStop : Bool := FALSE;   // TRUE = візок знаходиться в зоні технологічного передзупину назад
            ForwardPreStop : Bool := FALSE;   // TRUE = візок знаходиться в зоні технологічного передзупину вперед
            ForwardEncoderLimit : Bool := FALSE;   // TRUE = досягнута програмна межа по енкодеру вперед
            ForwardEmergencyLimit : Bool := FALSE;   // TRUE = досягнута позиція аварійного кінцевика вперед
            ForwardBuffer : Bool := FALSE;   // TRUE = досягнута або перевищена позиція буфера вперед
         END_STRUCT;
      END_STRUCT;
      Enc_4BR1 : Struct
         RawPoint1 : DInt := 1000000;   // Raw-значення, яке відповідає 0 мм.
         PositionPoint1_mm : LReal := 0.0;   // Перша координата, мм.
         RawPoint2 : DInt := 133_000_000;   // Raw-значення максимальної координати.
         PositionPoint2_mm : LReal := 11807.0;   // Максимальна координата за ТЗ. / Максимальна координата підйому за ТЗ.
         Position_mm : LReal := 893.489537075758;   // Поточне масштабоване положення.
         PositionRounded_mm : DInt := 893;   // Положення, округлене до цілого мм.
         PositionValid : Bool := TRUE;   // Положення придатне для штатного використання.
         CalculationValid : Bool := TRUE;   // Розрахунок виконано за достовірним raw.
         ConfigurationValid : Bool := TRUE;   // Контрольні точки задані коректно.
         InConfiguredRange : Bool := TRUE;   // Raw знаходиться між контрольними точками.
         BelowConfiguredRange : Bool := FALSE;   // Raw нижче налаштованого діапазону.
         AboveConfiguredRange : Bool := FALSE;   // Raw вище налаштованого діапазону.
         Scale_mm_per_count : LReal := 8.94469696969697E-05;   // Розрахований коефіцієнт масштабування.
         Status : Word := 16#0060;   // Діагностичне слово.
         ProgSwitches : Struct   // Програмні вимикачі
            LeftBuffer : Bool := FALSE;   // Досягнута позиція буфера зліва
            LeftEmergencyLimit : Bool := FALSE;   // Досягнута позиція аварійного кінцевика зліва
            LeftEncoderLimit : Bool := FALSE;   // Досягнута програмна межа по енкодеру зліва
            LeftPreStop : Bool := TRUE;   // Досягнута технологічна межа при русі вліво
            LeftZoneLimit : Bool := TRUE;   // Досягнута ліва межа зони
            RightZoneLimit : Bool := FALSE;   // Досягнута права межа зони
            RightPreStop : Bool := FALSE;   // Досягнута технологічна межа при русі вправо
            RightEncoderLimit : Bool := FALSE;   // Досягнута програмна межа по енкодеру справа
            RightEmergencyLimit : Bool := FALSE;   // Досягнута позиція аварійного кінцевика справа
            RightBuffer : Bool := FALSE;   // Досягнута позиція буфера справа
         END_STRUCT;
      END_STRUCT;
      Enc_4BR2 : Struct
         RawPoint1 : DInt := 200_000_000;   // Raw-значення, яке відповідає 0 мм.
         PositionPoint1_mm : LReal := 0.0;   // Перша координата, мм.
         RawPoint2 : DInt := 68000000;   // Raw-значення максимальної координати.
         PositionPoint2_mm : LReal := 11807.0;   // Максимальна координата за ТЗ. / Максимальна координата підйому за ТЗ.
         Position_mm : LReal := 893.480324037879;   // Поточне масштабоване положення.
         PositionRounded_mm : DInt := 893;   // Положення, округлене до цілого мм.
         PositionValid : Bool := TRUE;   // Положення придатне для штатного використання.
         CalculationValid : Bool := TRUE;   // Розрахунок виконано за достовірним raw.
         ConfigurationValid : Bool := TRUE;   // Контрольні точки задані коректно.
         InConfiguredRange : Bool := TRUE;   // Raw знаходиться між контрольними точками.
         BelowConfiguredRange : Bool := FALSE;   // Raw нижче налаштованого діапазону.
         AboveConfiguredRange : Bool := FALSE;   // Raw вище налаштованого діапазону.
         Scale_mm_per_count : LReal := -8.94469696969697E-05;   // Розрахований коефіцієнт масштабування.
         Status : Word := 16#0060;   // Діагностичне слово.
         ProgSwitches : Struct   // Програмні вимикачі
            LeftBuffer : Bool := FALSE;   // Досягнута позиція буфера зліва
            LeftEmergencyLimit : Bool := FALSE;   // Досягнута позиція аварійного кінцевика зліва
            LeftEncoderLimit : Bool := FALSE;   // Досягнута програмна межа по енкодеру зліва
            LeftPreStop : Bool := TRUE;   // Досягнута технологічна межа при русі вліво
            LeftZoneLimit : Bool := TRUE;   // Досягнута ліва межа зони
            RightZoneLimit : Bool := FALSE;   // Досягнута права межа зони
            RightPreStop : Bool := FALSE;   // Досягнута технологічна межа при русі вправо
            RightEncoderLimit : Bool := FALSE;   // Досягнута програмна межа по енкодеру справа
            RightEmergencyLimit : Bool := FALSE;   // Досягнута позиція аварійного кінцевика справа
            RightBuffer : Bool := FALSE;   // Досягнута позиція буфера справа
         END_STRUCT;
      END_STRUCT;
   END_VAR
BEGIN
END_DATA_BLOCK

DATA_BLOCK "DB_EncPositions"   // DB88
{ S7_Optimized_Access := 'TRUE' }
VERSION : 0.1
   VAR
      "1BR" : Struct   // Енкодер підйома
         DownEndPosition_mm : LReal := 0.0;   // Крайня нижня позиція механізму
         DownEmergencyLimit_mm : LReal := 50.0;   // Позиція аварійного кінцевика при опусканні
         DownEncoderLimit_mm : LReal := 200.0;   // Програмна межа по енкодеру при опусканні
         DownPreStop_mm : LReal := 700.0;   // Технологічний передзупин при опусканні
         UpPreStop_mm : LReal := 23500.0;   // Технологічний передзупин при підйомі
         UpEncoderLimit_mm : LReal := 23800.0;   // Програмна межа по енкодеру при підйомі
         UpEmergencyLimit_mm : LReal := 23950.0;   // Позиція аварійного кінцевика при підйомі
         UpEndPosition_mm : LReal := 24000.0;   // Крайня верхня позиція механізму
      END_STRUCT;
      "3BR" : Struct   // Енкодер візка
         BackBuffer_mm : LReal := 0.0;   // Крайня механічна позиція / буфер назад
         BackEmergencyLimit_mm : LReal := 50.0;   // Позиція аварійного апаратного кінцевика назад
         BackEncoderLimit_mm : LReal := 150.0;   // Програмна межа по енкодеру назад
         BackPreStop_mm : LReal := 900.0;   // Технологічний передзупин назад
         ForwardPreStop_mm : LReal := 7775.0;   // Технологічний передзупин вперед
         ForwardEncoderLimit_mm : LReal := 8525.0;   // Програмна межа по енкодеру вперед
         ForwardEmergencyLimit_mm : LReal := 8625.0;   // Позиція аварійного апаратного кінцевика вперед
         ForwardBuffer_mm : LReal := 8675.0;   // Крайня механічна позиція / буфер вперед
      END_STRUCT;
      "4BR1" : Struct   // Енкодер моста 1
         LeftBuffer_mm : LReal := 0.0;   // Позиція буфера зліва
         LeftEmergencyLimit_mm : LReal := 50.0;   // Позиція аварійного кінцевика зліва
         LeftEncoderLimit_mm : LReal := 150.0;   // Програмна межа по енкодеру зліва
         LeftPreStop_mm : LReal := 900.0;   // Технологічний передзупин при русі вліво
         LeftZoneLimit_mm : LReal := 3010.0;   // Ліва координатна межа зони
         RightZoneLimit_mm : LReal := 7125.0;   // Права координатна межа зони
         RightPreStop_mm : LReal := 10907.0;   // Технологічний передзупин при русі вправо
         RightEncoderLimit_mm : LReal := 11657.0;   // Програмна межа по енкодеру справа
         RightEmergencyLimit_mm : LReal := 11757.0;   // Позиція аварійного кінцевика справа
         RightBuffer_mm : LReal := 11807.0;   // Позиція буфера справа
      END_STRUCT;
      "4BR2" : Struct   // Енкодер моста 2
         LeftBuffer_mm : LReal := 0.0;   // Позиція буфера зліва
         LeftEmergencyLimit_mm : LReal := 50.0;   // Позиція аварійного кінцевика зліва
         LeftEncoderLimit_mm : LReal := 150.0;   // Програмна межа по енкодеру зліва
         LeftPreStop_mm : LReal := 900.0;   // Технологічний передзупин при русі вліво
         LeftZoneLimit_mm : LReal := 3010.0;   // Ліва координатна межа зони
         RightZoneLimit_mm : LReal := 7125.0;   // Права координатна межа зони
         RightPreStop_mm : LReal := 10907.0;   // Технологічний передзупин при русі вправо
         RightEncoderLimit_mm : LReal := 11657.0;   // Програмна межа по енкодеру справа
         RightEmergencyLimit_mm : LReal := 11757.0;   // Позиція аварійного кінцевика справа
         RightBuffer_mm : LReal := 11807.0;   // Позиція буфера справа
      END_STRUCT;
   END_VAR
BEGIN
END_DATA_BLOCK

DATA_BLOCK "DB_PosCorrection_1BR"   // DB90
{ S7_Optimized_Access := 'TRUE' }
VERSION : 0.1
// stored: InstanceOfName FB_PositionCorrection
"FB_PositionCorrection"
BEGIN
END_DATA_BLOCK

DATA_BLOCK "DB_PosCorrection_3BR"   // DB91
{ S7_Optimized_Access := 'TRUE' }
VERSION : 0.1
// stored: InstanceOfName FB_PositionCorrection
"FB_PositionCorrection"
BEGIN
END_DATA_BLOCK

DATA_BLOCK "DB_PosCorrection_4BR1"   // DB92
{ S7_Optimized_Access := 'TRUE' }
VERSION : 0.1
// stored: InstanceOfName FB_PositionCorrection
"FB_PositionCorrection"
BEGIN
END_DATA_BLOCK

DATA_BLOCK "DB_PosCorrection_4BR2"   // DB93
{ S7_Optimized_Access := 'TRUE' }
VERSION : 0.1
// stored: InstanceOfName FB_PositionCorrection
"FB_PositionCorrection"
BEGIN
END_DATA_BLOCK

// folder: System blocks/Program resources

DATA_BLOCK "IEC_Timer_0_DB"   // DB1002
{ S7_Optimized_Access := 'TRUE' }
AUTHOR : Simatic
FAMILY : IEC
NAME : IEC_TMR
VERSION : 1.0
// stored: InstanceOfName IEC_TIMER
"IEC_TIMER"
BEGIN
END_DATA_BLOCK

DATA_BLOCK "IEC_Timer_0_DB_1"   // DB1003
{ S7_Optimized_Access := 'TRUE' }
AUTHOR : Simatic
FAMILY : IEC
NAME : IEC_TMR
VERSION : 1.0
// stored: InstanceOfName IEC_TIMER
"IEC_TIMER"
BEGIN
END_DATA_BLOCK

DATA_BLOCK "IEC_Timer_0_DB_2"   // DB1004
{ S7_Optimized_Access := 'TRUE' }
AUTHOR : Simatic
FAMILY : IEC
NAME : IEC_TMR
VERSION : 1.0
// stored: InstanceOfName IEC_TIMER
"IEC_TIMER"
BEGIN
END_DATA_BLOCK

DATA_BLOCK "IEC_Timer_0_DB_3"   // DB1005
{ S7_Optimized_Access := 'TRUE' }
AUTHOR : Simatic
FAMILY : IEC
NAME : IEC_TMR
VERSION : 1.0
// stored: InstanceOfName IEC_TIMER
"IEC_TIMER"
BEGIN
END_DATA_BLOCK

DATA_BLOCK "IEC_Timer_0_DB_4"   // DB1006
{ S7_Optimized_Access := 'TRUE' }
AUTHOR : Simatic
FAMILY : IEC
NAME : IEC_TMR
VERSION : 1.0
// stored: InstanceOfName IEC_TIMER
"IEC_TIMER"
BEGIN
END_DATA_BLOCK

DATA_BLOCK "IEC_Timer_0_DB_5"   // DB1007
{ S7_Optimized_Access := 'TRUE' }
AUTHOR : Simatic
FAMILY : IEC
NAME : IEC_TMR
VERSION : 1.0
// stored: InstanceOfName IEC_TIMER
"IEC_TIMER"
BEGIN
END_DATA_BLOCK

DATA_BLOCK "IEC_Timer_0_DB_7"   // DB1009
{ S7_Optimized_Access := 'TRUE' }
AUTHOR : Simatic
FAMILY : IEC
NAME : IEC_TMR
VERSION : 1.0
// stored: InstanceOfName IEC_TIMER
"IEC_TIMER"
BEGIN
END_DATA_BLOCK

DATA_BLOCK "IEC_Timer_0_DB_8"   // DB1010
{ S7_Optimized_Access := 'TRUE' }
AUTHOR : Simatic
FAMILY : IEC
NAME : IEC_TMR
VERSION : 1.0
// stored: InstanceOfName IEC_TIMER
"IEC_TIMER"
BEGIN
END_DATA_BLOCK

DATA_BLOCK "IEC_Timer_0_DB_9"   // DB1011
{ S7_Optimized_Access := 'TRUE' }
AUTHOR : Simatic
FAMILY : IEC
NAME : IEC_TMR
VERSION : 1.0
// stored: InstanceOfName IEC_TIMER
"IEC_TIMER"
BEGIN
END_DATA_BLOCK

DATA_BLOCK "IEC_Timer_0_DB_10"   // DB1012
{ S7_Optimized_Access := 'TRUE' }
AUTHOR : Simatic
FAMILY : IEC
NAME : IEC_TMR
VERSION : 1.0
// stored: InstanceOfName IEC_TIMER
"IEC_TIMER"
BEGIN
END_DATA_BLOCK

DATA_BLOCK "IEC_Timer_DB_1BR"   // DB1201
{ S7_Optimized_Access := 'TRUE' }
AUTHOR : Simatic
FAMILY : IEC
NAME : IEC_TMR
VERSION : 1.0
// stored: InstanceOfName IEC_TIMER
"IEC_TIMER"
BEGIN
END_DATA_BLOCK

DATA_BLOCK "IEC_Timer_DB_3BR"   // DB1202
{ S7_Optimized_Access := 'TRUE' }
AUTHOR : Simatic
FAMILY : IEC
NAME : IEC_TMR
VERSION : 1.0
// stored: InstanceOfName IEC_TIMER
"IEC_TIMER"
BEGIN
END_DATA_BLOCK

DATA_BLOCK "IEC_Timer_DB_4BR"   // DB1203
{ S7_Optimized_Access := 'TRUE' }
AUTHOR : Simatic
FAMILY : IEC
NAME : IEC_TMR
VERSION : 1.0
// stored: InstanceOfName IEC_TIMER
"IEC_TIMER"
BEGIN
END_DATA_BLOCK

// folder: 0_OB

ORGANIZATION_BLOCK "Main"   // OB1, LAD, ProgramCycle
TITLE = "Main Program Sweep (Cycle)"
{ S7_Optimized_Access := 'TRUE' }
VERSION : 0.1
   VAR_INPUT
      Initial_Call : Bool;   // Initial call of this OB
      Remanence : Bool;   // =True, if remanent data are available
   END_VAR
   VAR_TEMP   // added for the SCL form of the ladder/FBD networks
      _w1 : Bool;
      _w2 : Bool;
   END_VAR
BEGIN

REGION Network 2: Setup (remove after abjustment)
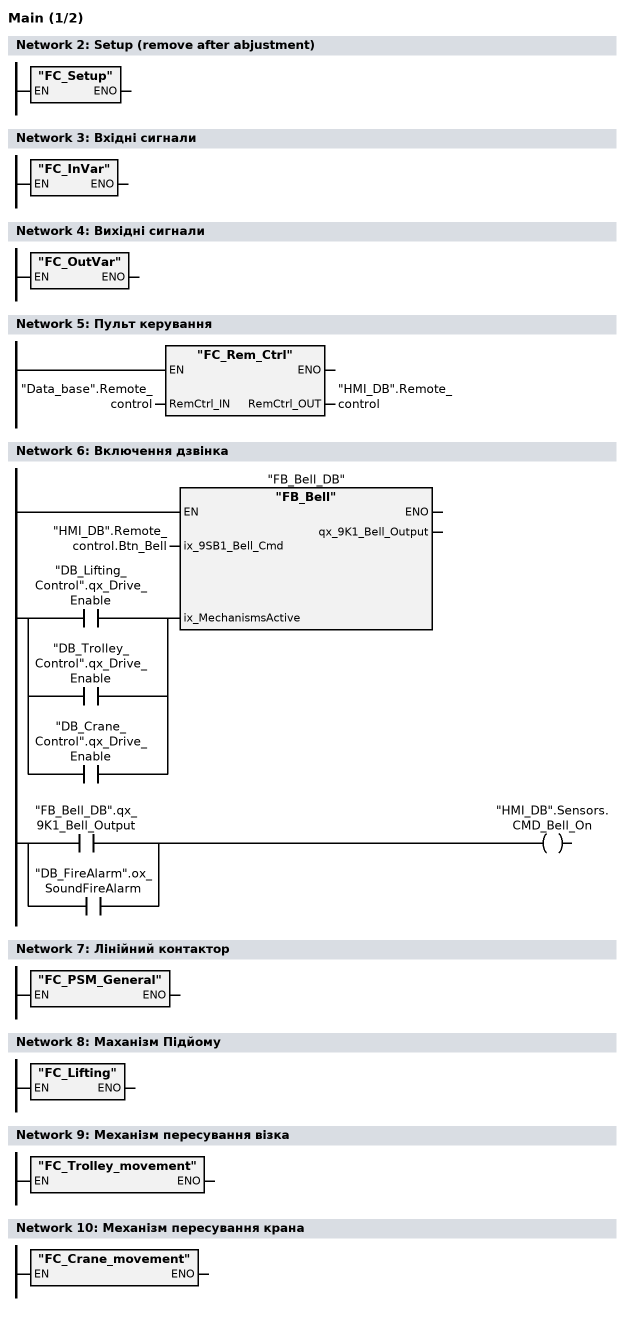
   RUNG wire#powerrail
      "FC_Setup"()
   END_RUNG
   // the same network as SCL:
   "FC_Setup"();
END_REGION

REGION Network 3: Вхідні сигнали
   RUNG wire#powerrail
      "FC_InVar"()
   END_RUNG
   // the same network as SCL:
   "FC_InVar"();
END_REGION

REGION Network 4: Вихідні сигнали
   RUNG wire#powerrail
      "FC_OutVar"()
   END_RUNG
   // the same network as SCL:
   "FC_OutVar"();
END_REGION

REGION Network 5: Пульт керування
   RUNG wire#powerrail
      "FC_Rem_Ctrl"(RemCtrl_IN := "Data_base".Remote_control, RemCtrl_OUT => "HMI_DB".Remote_control)
   END_RUNG
   // the same network as SCL:
   "FC_Rem_Ctrl"(RemCtrl_IN := "Data_base".Remote_control, RemCtrl_OUT => "HMI_DB".Remote_control);
END_REGION

REGION Network 6: Включення дзвінка
   RUNG wire#powerrail
      "FB_Bell_DB"(ix_MechanismsActive := wire#w1, ix_9SB1_Bell_Cmd := "HMI_DB".Remote_control.Btn_Bell, qx_9K1_Bell_Output =>)
   END_RUNG
   RUNG wire#powerrail
      Contact( "DB_Lifting_Control".qx_Drive_Enable )
   END_RUNG wire#w1
   RUNG wire#powerrail
      Contact( "DB_Trolley_Control".qx_Drive_Enable )
   END_RUNG wire#w1
   RUNG wire#powerrail
      Contact( "DB_Crane_Control".qx_Drive_Enable )
   END_RUNG wire#w1
   RUNG wire#powerrail
      Contact( "FB_Bell_DB".qx_9K1_Bell_Output )
      wire#w2
      Coil( "HMI_DB".Sensors.CMD_Bell_On )
   END_RUNG
   RUNG wire#powerrail
      Contact( "DB_FireAlarm".ox_SoundFireAlarm )
   END_RUNG wire#w2
   // the same network as SCL:
   "FB_Bell_DB"(ix_9SB1_Bell_Cmd := "HMI_DB".Remote_control.Btn_Bell,   // "FB_Bell"
                ix_MechanismsActive := "DB_Lifting_Control".qx_Drive_Enable OR "DB_Trolley_Control".qx_Drive_Enable OR "DB_Crane_Control".qx_Drive_Enable);
   "HMI_DB".Sensors.CMD_Bell_On := "FB_Bell_DB".qx_9K1_Bell_Output OR "DB_FireAlarm".ox_SoundFireAlarm;
END_REGION

REGION Network 7: Лінійний контактор
   RUNG wire#powerrail
      "FC_PSM_General"()
   END_RUNG
   // the same network as SCL:
   "FC_PSM_General"();
END_REGION

REGION Network 8: Маханізм Підйому
   RUNG wire#powerrail
      "FC_Lifting"()
   END_RUNG
   // the same network as SCL:
   "FC_Lifting"();
END_REGION

REGION Network 9: Механізм пересування візка
   RUNG wire#powerrail
      "FC_Trolley_movement"()
   END_RUNG
   // the same network as SCL:
   "FC_Trolley_movement"();
END_REGION

REGION Network 10: Механізм пересування крана
   RUNG wire#powerrail
      "FC_Crane_movement"()
   END_RUNG
   // the same network as SCL:
   "FC_Crane_movement"();
END_REGION

REGION Network 11: Encoders data to HMI
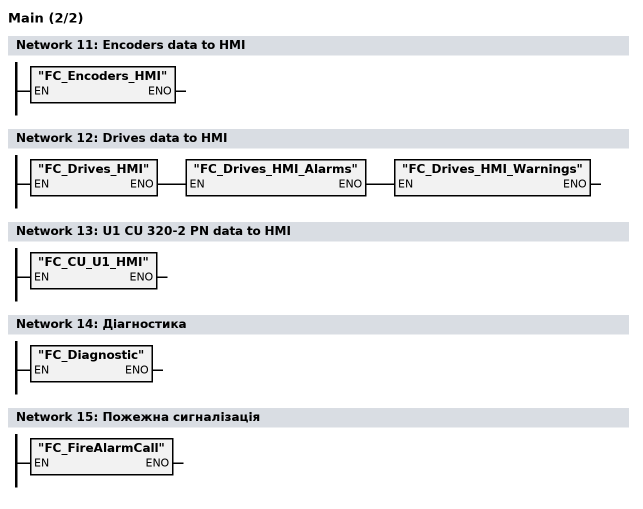
   RUNG wire#powerrail
      "FC_Encoders_HMI"()
   END_RUNG
   // the same network as SCL:
   "FC_Encoders_HMI"();
END_REGION

REGION Network 12: Drives data to HMI
   RUNG wire#powerrail
      "FC_Drives_HMI"()
      "FC_Drives_HMI_Alarms"()
      "FC_Drives_HMI_Warnings"()
   END_RUNG
   // the same network as SCL:
   "FC_Drives_HMI"(ENO => #_w1);
   "FC_Drives_HMI_Alarms"(EN := #_w1, ENO => #_w2);
   IF #_w2 THEN "FC_Drives_HMI_Warnings"(); END_IF;
END_REGION

REGION Network 13: U1 CU 320-2 PN data to HMI
   RUNG wire#powerrail
      "FC_CU_U1_HMI"()
   END_RUNG
   // the same network as SCL:
   "FC_CU_U1_HMI"();
END_REGION

REGION Network 14: Діагностика
   RUNG wire#powerrail
      "FC_Diagnostic"()
   END_RUNG
   // the same network as SCL:
   "FC_Diagnostic"();
END_REGION

REGION Network 15: Пожежна сигналізація
   RUNG wire#powerrail
      "FC_FireAlarmCall"()
   END_RUNG
   // the same network as SCL:
   "FC_FireAlarmCall"();
END_REGION
END_ORGANIZATION_BLOCK

ORGANIZATION_BLOCK "CyclicInterrupt"   // OB30, LAD, CyclicInterrupt
{ S7_Optimized_Access := 'TRUE' }
VERSION : 0.1
   VAR_INPUT
      Initial_Call : Bool;   // Initial call of this OB
      Event_Count : Int;   // Events discarded
   END_VAR
BEGIN

REGION Network 2: Комунікація з приводами
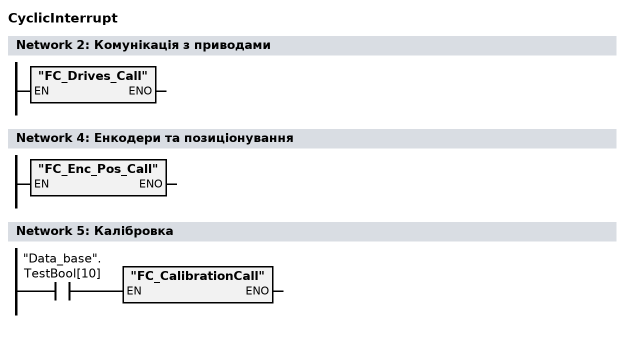
   RUNG wire#powerrail
      "FC_Drives_Call"()
   END_RUNG
   // the same network as SCL:
   "FC_Drives_Call"();
END_REGION

REGION Network 4: Енкодери та позиціонування
   RUNG wire#powerrail
      "FC_Enc_Pos_Call"()
   END_RUNG
   // the same network as SCL:
   "FC_Enc_Pos_Call"();
END_REGION

REGION Network 5: Калібровка
   RUNG wire#powerrail
      Contact( "Data_base".TestBool[10] )
      "FC_CalibrationCall"()
   END_RUNG
   // the same network as SCL:
   IF "Data_base".TestBool[10] THEN "FC_CalibrationCall"(); END_IF;
END_REGION
END_ORGANIZATION_BLOCK

// folder: 100_InOut

FUNCTION_BLOCK "FB_AnIn"   // FB100, LAD
{ S7_Optimized_Access := 'TRUE' }
VERSION : 0.1
   VAR_INPUT
      iiVRaw : Int;   // Raw value (from input channel)
   END_VAR
   VAR_OUTPUT
      orVal : Real;   // Output value
   END_VAR
   VAR_IN_OUT
      VarCfg : "AnICfg";   // Analog input variable
   END_VAR
   VAR
      VAL : Real;   // Intermediate value
      FB_StateDefine_LO : "FB_StateDefine";
      FB_StateDefine_LOLO : "FB_StateDefine";
      FB_StateDefine_HI : "FB_StateDefine";
      FB_StateDefine_HIHI : "FB_StateDefine";
      LORaw : Int := -27648;   // Raw value LO limit
      HIRaw : Int := 27648;   // Raw value HI limit
      LOPhy : Real := -10.0;   // Physical value LO limit (mA)
      HIPhy : Real := 10.0;   // Physical value HI limit (mA)
      FltScale : Bool;   // Fault scale
   END_VAR
   VAR_TEMP
      Temp1 : Real;
   END_VAR
   VAR_TEMP   // added for the SCL form of the ladder/FBD networks
      _w1 : Bool;
   END_VAR
BEGIN

REGION Network 1: Input modul value
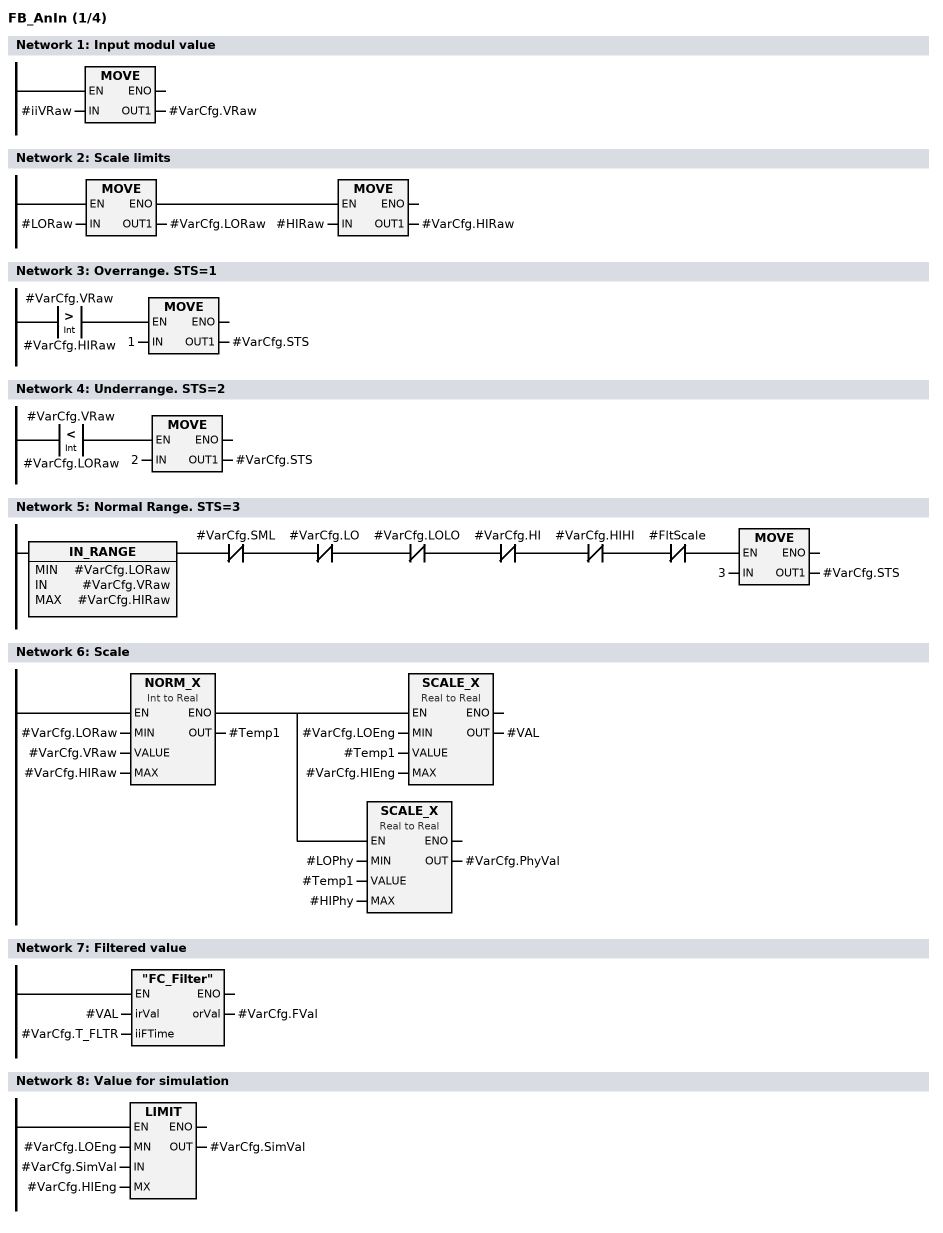
   RUNG wire#powerrail
      Move(in := #iiVRaw, out1 => #VarCfg.VRaw)
   END_RUNG
   // the same network as SCL:
   #VarCfg.VRaw := #iiVRaw;
END_REGION

REGION Network 2: Scale limits
   RUNG wire#powerrail
      Move(in := #LORaw, out1 => #VarCfg.LORaw)
      Move(in := #HIRaw, out1 => #VarCfg.HIRaw)
   END_RUNG
   // the same network as SCL:
   #VarCfg.LORaw := #LORaw;
   #VarCfg.HIRaw := #HIRaw;
END_REGION

REGION Network 3: Overrange. STS=1
   RUNG wire#powerrail
      { S7_Templates := "SrcType := Int" } GT_Contact(in1 := #VarCfg.VRaw, in2 := #VarCfg.HIRaw)
      Move(in := 1, out1 => #VarCfg.STS)
   END_RUNG
   // the same network as SCL:
   IF #VarCfg.VRaw > #VarCfg.HIRaw THEN #VarCfg.STS := 1; END_IF;
END_REGION

REGION Network 4: Underrange. STS=2
   RUNG wire#powerrail
      { S7_Templates := "SrcType := Int" } LT_Contact(in1 := #VarCfg.VRaw, in2 := #VarCfg.LORaw)
      Move(in := 2, out1 => #VarCfg.STS)
   END_RUNG
   // the same network as SCL:
   IF #VarCfg.VRaw < #VarCfg.LORaw THEN #VarCfg.STS := 2; END_IF;
END_REGION

REGION Network 5: Normal Range. STS=3
   RUNG wire#powerrail
      { S7_Templates := "SrcType := Int" } InRange(min := #VarCfg.LORaw, in := #VarCfg.VRaw, max := #VarCfg.HIRaw)
      I_Contact( #VarCfg.SML )
      I_Contact( #VarCfg.LO )
      I_Contact( #VarCfg.LOLO )
      I_Contact( #VarCfg.HI )
      I_Contact( #VarCfg.HIHI )
      I_Contact( #FltScale )
      Move(in := 3, out1 => #VarCfg.STS)
   END_RUNG
   // the same network as SCL:
   IF (#VarCfg.LORaw <= #VarCfg.VRaw) AND (#VarCfg.VRaw <= #VarCfg.HIRaw) AND NOT #VarCfg.SML AND NOT #VarCfg.LO AND NOT #VarCfg.LOLO AND NOT #VarCfg.HI AND NOT #VarCfg.HIHI AND NOT #FltScale THEN
       #VarCfg.STS := 3;
   END_IF;
END_REGION

REGION Network 6: Scale
   RUNG wire#powerrail
      { S7_Templates := "[SrcType := Int, DestType := Real]" } Normalize(min := #VarCfg.LORaw, value := #VarCfg.VRaw, max := #VarCfg.HIRaw, out => #Temp1)
      wire#w1
      { S7_Templates := "[SrcType := Real, DestType := Real]" } Scale(min := #VarCfg.LOEng, value := #Temp1, max := #VarCfg.HIEng, out => #VAL)
   END_RUNG
   RUNG wire#w1
      { S7_Templates := "[SrcType := Real, DestType := Real]" } Scale(min := #LOPhy, value := #Temp1, max := #HIPhy, out => #VarCfg.PhyVal)
   END_RUNG
   // the same network as SCL:
   #Temp1 := NORM_X(MIN := #VarCfg.LORaw, VALUE := #VarCfg.VRaw, MAX := #VarCfg.HIRaw);
   #VAL := SCALE_X(MIN := #VarCfg.LOEng, VALUE := #Temp1, MAX := #VarCfg.HIEng);
   #VarCfg.PhyVal := SCALE_X(MIN := #LOPhy, VALUE := #Temp1, MAX := #HIPhy);
END_REGION

REGION Network 7: Filtered value
   RUNG wire#powerrail
      "FC_Filter"(irVal := #VAL, iiFTime := #VarCfg.T_FLTR, orVal => #VarCfg.FVal)
   END_RUNG
   // the same network as SCL:
   "FC_Filter"(irVal := #VAL, iiFTime := #VarCfg.T_FLTR, orVal => #VarCfg.FVal);
END_REGION

REGION Network 8: Value for simulation
   #VarCfg.SimVal := LIMIT(MN := #VarCfg.LOEng, IN := #VarCfg.SimVal, MX := #VarCfg.HIEng);
END_REGION

REGION Network 9: Output value is simulated
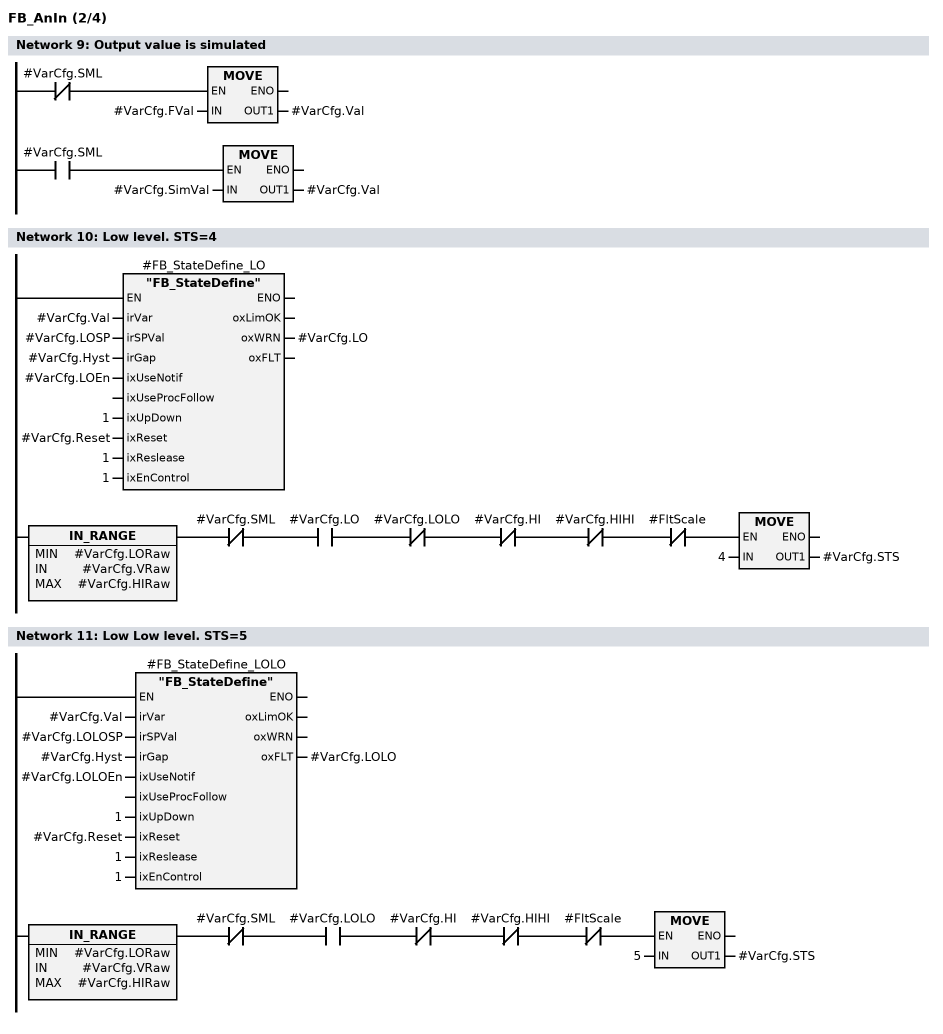
   RUNG wire#powerrail
      I_Contact( #VarCfg.SML )
      Move(in := #VarCfg.FVal, out1 => #VarCfg.Val)
   END_RUNG
   RUNG wire#powerrail
      Contact( #VarCfg.SML )
      Move(in := #VarCfg.SimVal, out1 => #VarCfg.Val)
   END_RUNG
   // the same network as SCL:
   IF NOT #VarCfg.SML THEN #VarCfg.Val := #VarCfg.FVal; END_IF;
   IF #VarCfg.SML THEN #VarCfg.Val := #VarCfg.SimVal; END_IF;
END_REGION

REGION Network 10: Low level. STS=4
   RUNG wire#powerrail
      #FB_StateDefine_LO(irVar := #VarCfg.Val, irSPVal := #VarCfg.LOSP, irGap := #VarCfg.Hyst, ixUseNotif := #VarCfg.LOEn, ixUseProcFollow :=, ixUpDown := 1, ixReset := #VarCfg.Reset, ixReslease := 1, ixEnControl := 1, oxLimOK =>, oxWRN => #VarCfg.LO, oxFLT =>)
   END_RUNG
   RUNG wire#powerrail
      { S7_Templates := "SrcType := Int" } InRange(min := #VarCfg.LORaw, in := #VarCfg.VRaw, max := #VarCfg.HIRaw)
      I_Contact( #VarCfg.SML )
      Contact( #VarCfg.LO )
      I_Contact( #VarCfg.LOLO )
      I_Contact( #VarCfg.HI )
      I_Contact( #VarCfg.HIHI )
      I_Contact( #FltScale )
      Move(in := 4, out1 => #VarCfg.STS)
   END_RUNG
   // the same network as SCL:
   #FB_StateDefine_LO(irVar := #VarCfg.Val,   // "FB_StateDefine"
                      irSPVal := #VarCfg.LOSP,
                      irGap := #VarCfg.Hyst,
                      ixUseNotif := #VarCfg.LOEn,
                      ixUpDown := 1,
                      ixReset := #VarCfg.Reset,
                      ixReslease := 1,
                      ixEnControl := 1,
                      oxWRN => #VarCfg.LO);
   IF (#VarCfg.LORaw <= #VarCfg.VRaw) AND (#VarCfg.VRaw <= #VarCfg.HIRaw) AND NOT #VarCfg.SML AND #VarCfg.LO AND NOT #VarCfg.LOLO AND NOT #VarCfg.HI AND NOT #VarCfg.HIHI AND NOT #FltScale THEN
       #VarCfg.STS := 4;
   END_IF;
END_REGION

REGION Network 11: Low Low level. STS=5
   RUNG wire#powerrail
      #FB_StateDefine_LOLO(irVar := #VarCfg.Val, irSPVal := #VarCfg.LOLOSP, irGap := #VarCfg.Hyst, ixUseNotif := #VarCfg.LOLOEn, ixUseProcFollow :=, ixUpDown := 1, ixReset := #VarCfg.Reset, ixReslease := 1, ixEnControl := 1, oxLimOK =>, oxWRN =>, oxFLT => #VarCfg.LOLO)
   END_RUNG
   RUNG wire#powerrail
      { S7_Templates := "SrcType := Int" } InRange(min := #VarCfg.LORaw, in := #VarCfg.VRaw, max := #VarCfg.HIRaw)
      I_Contact( #VarCfg.SML )
      Contact( #VarCfg.LOLO )
      I_Contact( #VarCfg.HI )
      I_Contact( #VarCfg.HIHI )
      I_Contact( #FltScale )
      Move(in := 5, out1 => #VarCfg.STS)
   END_RUNG
   // the same network as SCL:
   #FB_StateDefine_LOLO(irVar := #VarCfg.Val,   // "FB_StateDefine"
                        irSPVal := #VarCfg.LOLOSP,
                        irGap := #VarCfg.Hyst,
                        ixUseNotif := #VarCfg.LOLOEn,
                        ixUpDown := 1,
                        ixReset := #VarCfg.Reset,
                        ixReslease := 1,
                        ixEnControl := 1,
                        oxFLT => #VarCfg.LOLO);
   IF (#VarCfg.LORaw <= #VarCfg.VRaw) AND (#VarCfg.VRaw <= #VarCfg.HIRaw) AND NOT #VarCfg.SML AND #VarCfg.LOLO AND NOT #VarCfg.HI AND NOT #VarCfg.HIHI AND NOT #FltScale THEN
       #VarCfg.STS := 5;
   END_IF;
END_REGION

REGION Network 12: High level. STS=6
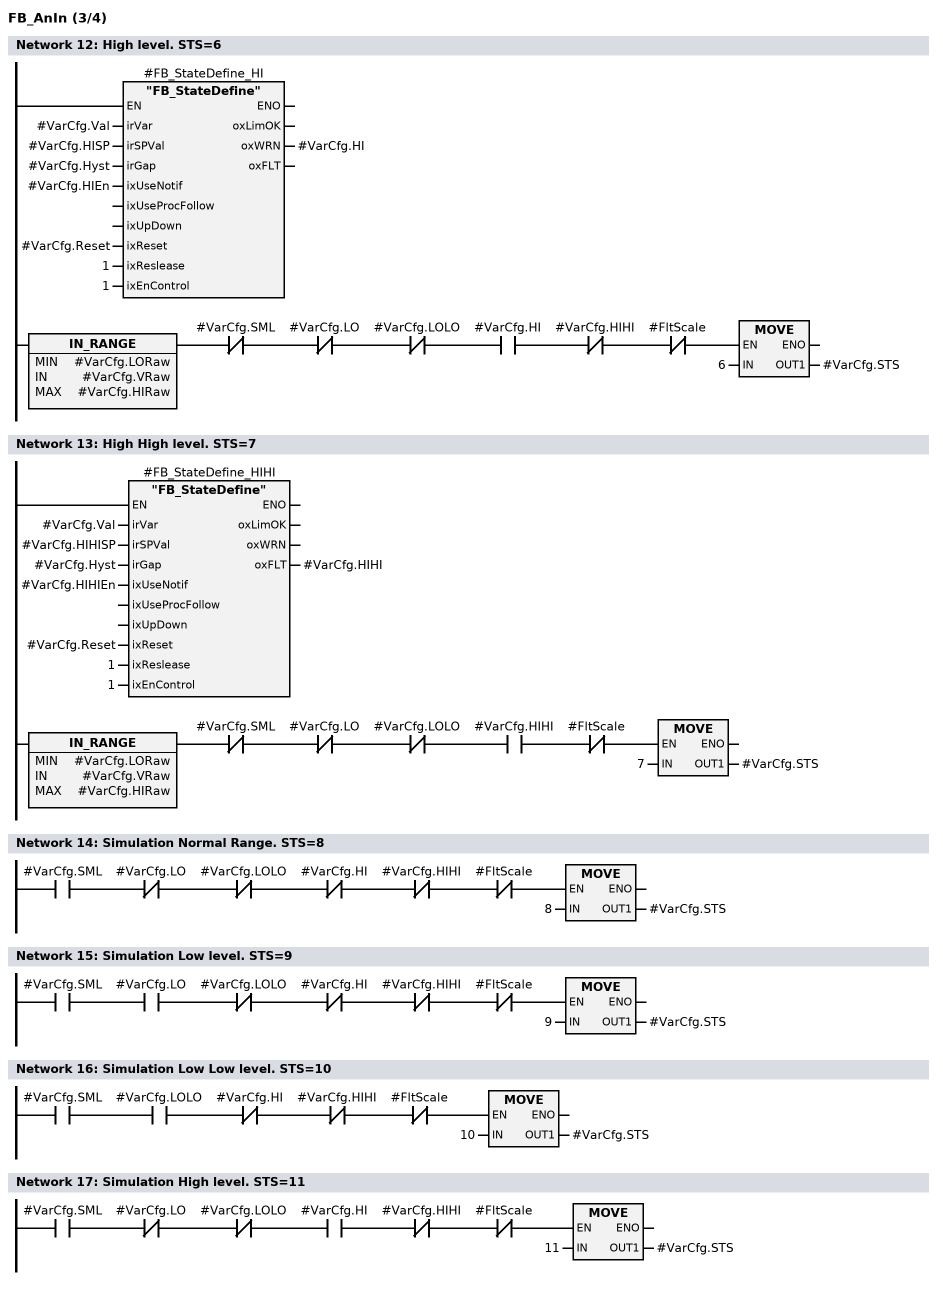
   RUNG wire#powerrail
      #FB_StateDefine_HI(irVar := #VarCfg.Val, irSPVal := #VarCfg.HISP, irGap := #VarCfg.Hyst, ixUseNotif := #VarCfg.HIEn, ixUseProcFollow :=, ixUpDown :=, ixReset := #VarCfg.Reset, ixReslease := 1, ixEnControl := 1, oxLimOK =>, oxWRN => #VarCfg.HI, oxFLT =>)
   END_RUNG
   RUNG wire#powerrail
      { S7_Templates := "SrcType := Int" } InRange(min := #VarCfg.LORaw, in := #VarCfg.VRaw, max := #VarCfg.HIRaw)
      I_Contact( #VarCfg.SML )
      I_Contact( #VarCfg.LO )
      I_Contact( #VarCfg.LOLO )
      Contact( #VarCfg.HI )
      I_Contact( #VarCfg.HIHI )
      I_Contact( #FltScale )
      Move(in := 6, out1 => #VarCfg.STS)
   END_RUNG
   // the same network as SCL:
   #FB_StateDefine_HI(irVar := #VarCfg.Val,   // "FB_StateDefine"
                      irSPVal := #VarCfg.HISP,
                      irGap := #VarCfg.Hyst,
                      ixUseNotif := #VarCfg.HIEn,
                      ixReset := #VarCfg.Reset,
                      ixReslease := 1,
                      ixEnControl := 1,
                      oxWRN => #VarCfg.HI);
   IF (#VarCfg.LORaw <= #VarCfg.VRaw) AND (#VarCfg.VRaw <= #VarCfg.HIRaw) AND NOT #VarCfg.SML AND NOT #VarCfg.LO AND NOT #VarCfg.LOLO AND #VarCfg.HI AND NOT #VarCfg.HIHI AND NOT #FltScale THEN
       #VarCfg.STS := 6;
   END_IF;
END_REGION

REGION Network 13: High High level. STS=7
   RUNG wire#powerrail
      #FB_StateDefine_HIHI(irVar := #VarCfg.Val, irSPVal := #VarCfg.HIHISP, irGap := #VarCfg.Hyst, ixUseNotif := #VarCfg.HIHIEn, ixUseProcFollow :=, ixUpDown :=, ixReset := #VarCfg.Reset, ixReslease := 1, ixEnControl := 1, oxLimOK =>, oxWRN =>, oxFLT => #VarCfg.HIHI)
   END_RUNG
   RUNG wire#powerrail
      { S7_Templates := "SrcType := Int" } InRange(min := #VarCfg.LORaw, in := #VarCfg.VRaw, max := #VarCfg.HIRaw)
      I_Contact( #VarCfg.SML )
      I_Contact( #VarCfg.LO )
      I_Contact( #VarCfg.LOLO )
      Contact( #VarCfg.HIHI )
      I_Contact( #FltScale )
      Move(in := 7, out1 => #VarCfg.STS)
   END_RUNG
   // the same network as SCL:
   #FB_StateDefine_HIHI(irVar := #VarCfg.Val,   // "FB_StateDefine"
                        irSPVal := #VarCfg.HIHISP,
                        irGap := #VarCfg.Hyst,
                        ixUseNotif := #VarCfg.HIHIEn,
                        ixReset := #VarCfg.Reset,
                        ixReslease := 1,
                        ixEnControl := 1,
                        oxFLT => #VarCfg.HIHI);
   IF (#VarCfg.LORaw <= #VarCfg.VRaw) AND (#VarCfg.VRaw <= #VarCfg.HIRaw) AND NOT #VarCfg.SML AND NOT #VarCfg.LO AND NOT #VarCfg.LOLO AND #VarCfg.HIHI AND NOT #FltScale THEN
       #VarCfg.STS := 7;
   END_IF;
END_REGION

REGION Network 14: Simulation Normal Range. STS=8
   RUNG wire#powerrail
      Contact( #VarCfg.SML )
      I_Contact( #VarCfg.LO )
      I_Contact( #VarCfg.LOLO )
      I_Contact( #VarCfg.HI )
      I_Contact( #VarCfg.HIHI )
      I_Contact( #FltScale )
      Move(in := 8, out1 => #VarCfg.STS)
   END_RUNG
   // the same network as SCL:
   IF #VarCfg.SML AND NOT #VarCfg.LO AND NOT #VarCfg.LOLO AND NOT #VarCfg.HI AND NOT #VarCfg.HIHI AND NOT #FltScale THEN
       #VarCfg.STS := 8;
   END_IF;
END_REGION

REGION Network 15: Simulation Low level. STS=9
   RUNG wire#powerrail
      Contact( #VarCfg.SML )
      Contact( #VarCfg.LO )
      I_Contact( #VarCfg.LOLO )
      I_Contact( #VarCfg.HI )
      I_Contact( #VarCfg.HIHI )
      I_Contact( #FltScale )
      Move(in := 9, out1 => #VarCfg.STS)
   END_RUNG
   // the same network as SCL:
   IF #VarCfg.SML AND #VarCfg.LO AND NOT #VarCfg.LOLO AND NOT #VarCfg.HI AND NOT #VarCfg.HIHI AND NOT #FltScale THEN
       #VarCfg.STS := 9;
   END_IF;
END_REGION

REGION Network 16: Simulation Low Low level. STS=10
   RUNG wire#powerrail
      Contact( #VarCfg.SML )
      Contact( #VarCfg.LOLO )
      I_Contact( #VarCfg.HI )
      I_Contact( #VarCfg.HIHI )
      I_Contact( #FltScale )
      Move(in := 10, out1 => #VarCfg.STS)
   END_RUNG
   // the same network as SCL:
   IF #VarCfg.SML AND #VarCfg.LOLO AND NOT #VarCfg.HI AND NOT #VarCfg.HIHI AND NOT #FltScale THEN
       #VarCfg.STS := 10;
   END_IF;
END_REGION

REGION Network 17: Simulation High level. STS=11
   RUNG wire#powerrail
      Contact( #VarCfg.SML )
      I_Contact( #VarCfg.LO )
      I_Contact( #VarCfg.LOLO )
      Contact( #VarCfg.HI )
      I_Contact( #VarCfg.HIHI )
      I_Contact( #FltScale )
      Move(in := 11, out1 => #VarCfg.STS)
   END_RUNG
   // the same network as SCL:
   IF #VarCfg.SML AND NOT #VarCfg.LO AND NOT #VarCfg.LOLO AND #VarCfg.HI AND NOT #VarCfg.HIHI AND NOT #FltScale THEN
       #VarCfg.STS := 11;
   END_IF;
END_REGION

REGION Network 18: Simulation High level. STS=12
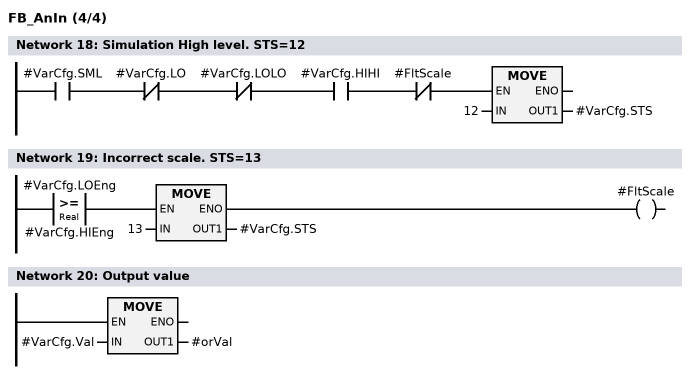
   RUNG wire#powerrail
      Contact( #VarCfg.SML )
      I_Contact( #VarCfg.LO )
      I_Contact( #VarCfg.LOLO )
      Contact( #VarCfg.HIHI )
      I_Contact( #FltScale )
      Move(in := 12, out1 => #VarCfg.STS)
   END_RUNG
   // the same network as SCL:
   IF #VarCfg.SML AND NOT #VarCfg.LO AND NOT #VarCfg.LOLO AND #VarCfg.HIHI AND NOT #FltScale THEN
       #VarCfg.STS := 12;
   END_IF;
END_REGION

REGION Network 19: Incorrect scale. STS=13
   RUNG wire#powerrail
      { S7_Templates := "SrcType := Real" } GE_Contact(in1 := #VarCfg.LOEng, in2 := #VarCfg.HIEng)
      Move(in := 13, out1 => #VarCfg.STS)
      Coil( #FltScale )
   END_RUNG
   // the same network as SCL:
   #_w1 := #VarCfg.LOEng >= #VarCfg.HIEng;
   IF #_w1 THEN #VarCfg.STS := 13; END_IF;
   #FltScale := #_w1;
END_REGION

REGION Network 20: Output value
   RUNG wire#powerrail
      Move(in := #VarCfg.Val, out1 => #orVal)
   END_RUNG
   // the same network as SCL:
   #orVal := #VarCfg.Val;
END_REGION
END_FUNCTION_BLOCK

FUNCTION_BLOCK "FB_DigIn"   // FB101, LAD
{ S7_Optimized_Access := 'TRUE' }
VERSION : 0.1
   VAR_INPUT
      ixVRaw : Bool;   // RAW value
   END_VAR
   VAR_OUTPUT
      oxVal : Bool;   // Processed signal
   END_VAR
   VAR_IN_OUT
      VarCfg : "DigICfg";   // Discrete input variable
   END_VAR
BEGIN

REGION Network 1: RAW value
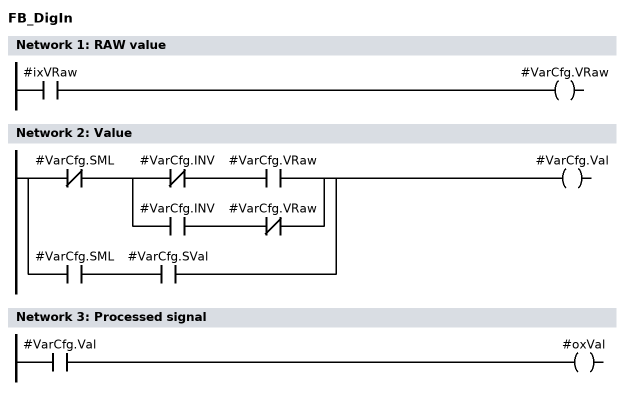
   RUNG wire#powerrail
      Contact( #ixVRaw )
      Coil( #VarCfg.VRaw )
   END_RUNG
   // the same network as SCL:
   #VarCfg.VRaw := #ixVRaw;
END_REGION

REGION Network 2: Value
   RUNG wire#powerrail
      I_Contact( #VarCfg.SML )
      wire#w1
      I_Contact( #VarCfg.INV )
      Contact( #VarCfg.VRaw )
      wire#w2
      Coil( #VarCfg.Val )
   END_RUNG
   RUNG wire#w1
      Contact( #VarCfg.INV )
      I_Contact( #VarCfg.VRaw )
   END_RUNG wire#w2
   RUNG wire#powerrail
      Contact( #VarCfg.SML )
      Contact( #VarCfg.SVal )
   END_RUNG wire#w2
   // the same network as SCL:
   #VarCfg.Val := (NOT #VarCfg.SML AND ((NOT #VarCfg.INV AND #VarCfg.VRaw) OR (#VarCfg.INV AND NOT #VarCfg.VRaw))) OR (#VarCfg.SML AND #VarCfg.SVal);
END_REGION

REGION Network 3: Processed signal
   RUNG wire#powerrail
      Contact( #VarCfg.Val )
      Coil( #oxVal )
   END_RUNG
   // the same network as SCL:
   #oxVal := #VarCfg.Val;
END_REGION
END_FUNCTION_BLOCK

FUNCTION_BLOCK "FB_DigOut"   // FB102, LAD
{ S7_Optimized_Access := 'TRUE' }
VERSION : 0.1
   VAR_INPUT
      ixVRaw : Bool;   // RAW value
   END_VAR
   VAR_OUTPUT
      oxVal : Bool;   // Processed signal
   END_VAR
   VAR_IN_OUT
      VarCfg : "DigOCfg";   // Discrete output variable
   END_VAR
BEGIN

REGION Network 1: RAW value
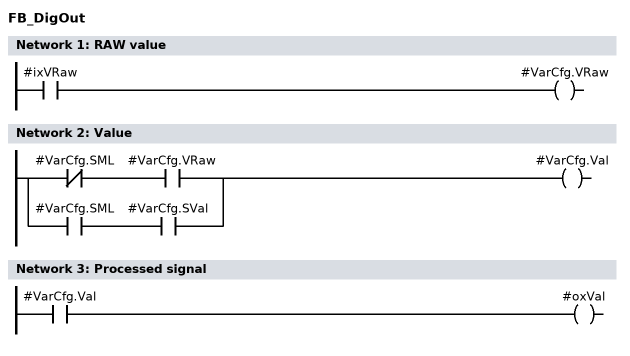
   RUNG wire#powerrail
      Contact( #ixVRaw )
      Coil( #VarCfg.VRaw )
   END_RUNG
   // the same network as SCL:
   #VarCfg.VRaw := #ixVRaw;
END_REGION

REGION Network 2: Value
   RUNG wire#powerrail
      I_Contact( #VarCfg.SML )
      Contact( #VarCfg.VRaw )
      wire#w1
      Coil( #VarCfg.Val )
   END_RUNG
   RUNG wire#powerrail
      Contact( #VarCfg.SML )
      Contact( #VarCfg.SVal )
   END_RUNG wire#w1
   // the same network as SCL:
   #VarCfg.Val := (NOT #VarCfg.SML AND #VarCfg.VRaw) OR (#VarCfg.SML AND #VarCfg.SVal);
END_REGION

REGION Network 3: Processed signal
   RUNG wire#powerrail
      Contact( #VarCfg.Val )
      Coil( #oxVal )
   END_RUNG
   // the same network as SCL:
   #oxVal := #VarCfg.Val;
END_REGION
END_FUNCTION_BLOCK

FUNCTION "FC_InVar" : Void   // FC100, SCL
TITLE = Inputs
{ S7_Optimized_Access := 'TRUE' }
AUTHOR : DZH
VERSION : 0.1
// Controller Discrete and Analog Inputs
BEGIN
   REGION KZPTO
   REGION A1_2

           "DB_DigIn_I0.0"(ixVRaw:="6KM1", oxVal=>"HMI_DB".PSM.Line_contactor_On, VarCfg:="HMI_DB".IO_Tags.InCnf.DigIn_0_0);
           "DB_DigIn_I0.1"(ixVRaw:="6KM2", oxVal=>"HMI_DB".PSM.Control_contactor_220V_On, VarCfg:="HMI_DB".IO_Tags.InCnf.DigIn_0_1);
           "DB_DigIn_I0.2"(ixVRaw:="6KV", oxVal=>"HMI_DB".PSM.Input_voltage_control_380V_On, VarCfg:="HMI_DB".IO_Tags.InCnf.DigIn_0_2);
           "DB_DigIn_I0.3"(ixVRaw:="6SF5", oxVal=>"HMI_DB".PSM.Heating_circuit_breaker_220V_On,VarCfg:="HMI_DB".IO_Tags.InCnf.DigIn_0_3);
           "DB_DigIn_I0.4"(ixVRaw:="6QF2", oxVal=> "HMI_DB".PSM.Brake_protection_On,VarCfg:="HMI_DB".IO_Tags.InCnf.DigIn_0_4);
           "DB_DigIn_I0.5"(ixVRaw:="6QF3", oxVal=> "HMI_DB".PSM.Transformer_6T1_380V_On,VarCfg:="HMI_DB".IO_Tags.InCnf.DigIn_0_5);
           "DB_DigIn_I0.6"(ixVRaw:="6QF4", oxVal=>"HMI_DB".PSM.Transformer_sec_circuit_breaker_6T1_380V_On,VarCfg:="HMI_DB".IO_Tags.InCnf.DigIn_0_6);
           "DB_DigIn_I0.7"(ixVRaw:="6SF1", oxVal=> "HMI_DB".PSM.Power_switch_6KV_380V_On,VarCfg:="HMI_DB".IO_Tags.InCnf.DigIn_0_7);
           "DB_DigIn_I1.0"(ixVRaw:="6SF2", oxVal=>"HMI_DB".PSM.ID_Control_circuit_breaker_220V_On,VarCfg:="HMI_DB".IO_Tags.InCnf.DigIn_1_0);
           "DB_DigIn_I1.1"(ixVRaw:="6SF4", oxVal=>"HMI_DB".PSM.ID_ORP_power_circuit_breaker_220V_On,VarCfg:="HMI_DB".IO_Tags.InCnf.DigIn_1_1);
           "DB_DigIn_I1.2"(ixVRaw:="6K3", oxVal=>"HMI_DB".PSM.ID_Line_contactor_from_remote_control_On,VarCfg:="HMI_DB".IO_Tags.InCnf.DigIn_1_2);
           "DB_DigIn_I1.3"(ixVRaw:="9QF2", oxVal=>"HMI_DB".PSM.Transformer_9T1_380V_On,VarCfg:="HMI_DB".IO_Tags.InCnf.DigIn_1_3);
           "DB_DigIn_I1.4"(ixVRaw:="9QF3", oxVal=>"HMI_DB".PSM.Repair_lighting_switch_12V_On, VarCfg:="HMI_DB".IO_Tags.InCnf.DigIn_1_4);
           "DB_DigIn_I1.5"(ixVRaw:="9QF4", oxVal=>"HMI_DB".PSM.Cabinet_circuit_breaker_220V_On,VarCfg:="HMI_DB".IO_Tags.InCnf.DigIn_1_5);
           "DB_DigIn_I1.6"(ixVRaw:="9K2", oxVal=>"HMI_DB".Sensors.Cabinet_heating_control_SU1,VarCfg:="HMI_DB".IO_Tags.InCnf.DigIn_1_6);
           "DB_DigIn_I1.7"(ixVRaw:="9K3", oxVal=>"HMI_DB".Sensors.Seismic_sensor,VarCfg:="HMI_DB".IO_Tags.InCnf.DigIn_1_7);
           "DB_DigIn_I2.0"(ixVRaw:="S1_Up", oxVal=>"Data_base".Remote_control.Btn_Up,VarCfg:="HMI_DB".IO_Tags.InCnf.DigIn_2_0);
           "DB_DigIn_I2.1"(ixVRaw:="S1_Down", oxVal=>"Data_base".Remote_control.Btn_Down,VarCfg:="HMI_DB".IO_Tags.InCnf.DigIn_2_1);
           "DB_DigIn_I2.2"(ixVRaw:="S1_Forward", oxVal=>"Data_base".Remote_control.Btn_Fwd,VarCfg:="HMI_DB".IO_Tags.InCnf.DigIn_2_2);
           "DB_DigIn_I2.3"(ixVRaw:="S1_Backward", oxVal=>"Data_base".Remote_control.Btn_Bwd,VarCfg:="HMI_DB".IO_Tags.InCnf.DigIn_2_3);
           "DB_DigIn_I2.4"(ixVRaw:="S1_Left", oxVal=>"Data_base".Remote_control.Btn_Left,VarCfg:="HMI_DB".IO_Tags.InCnf.DigIn_2_4);
           "DB_DigIn_I2.5"(ixVRaw:="S1_Right", oxVal=>"Data_base".Remote_control.Btn_Right,VarCfg:="HMI_DB".IO_Tags.InCnf.DigIn_2_5);
           "DB_DigIn_I2.6"(ixVRaw:="S2_Speed", oxVal=>"Data_base".Remote_control.Btn_ScndSpeed,VarCfg:="HMI_DB".IO_Tags.InCnf.DigIn_2_6);
           "DB_DigIn_I2.7"(ixVRaw:="Bell", oxVal=>"Data_base".Remote_control.Btn_Bell,VarCfg:="HMI_DB".IO_Tags.InCnf.DigIn_2_7);
           "DB_DigIn_I3.0"(ixVRaw:="I3_0", oxVal=>"HMI_DB".Reserv.I3_0,VarCfg:="HMI_DB".IO_Tags.InCnf.DigIn_3_0);
           "DB_DigIn_I3.1"(ixVRaw:="1BV", oxVal=>"HMI_DB".Sensors.Drum_rotation_control,VarCfg:="HMI_DB".IO_Tags.InCnf.DigIn_3_1);
           "DB_DigIn_I3.2"(ixVRaw:="1BM1_Up", oxVal=>"HMI_DB".Lifting_mechanism.Work_control,VarCfg:="HMI_DB".IO_Tags.InCnf.DigIn_3_2);
           "DB_DigIn_I3.3"(ixVRaw:="1BM1_Brake", oxVal=>"HMI_DB".Lifting_mechanism.Brake_wear_control,VarCfg:="HMI_DB".IO_Tags.InCnf.DigIn_3_3);
           "DB_DigIn_I3.4"(ixVRaw:="1K41", oxVal=>"HMI_DB".Lifting_mechanism.MD_disconnected_from_drive,VarCfg:="HMI_DB".IO_Tags.InCnf.DigIn_3_4);
           "DB_DigIn_I3.5"(ixVRaw:="4QF1", oxVal=>"HMI_DB".Crane_movement_mechanism.Brake_protection_On,VarCfg:="HMI_DB".IO_Tags.InCnf.DigIn_3_5);
           "DB_DigIn_I3.6"(ixVRaw:="4KT1", oxVal=>"HMI_DB".Crane_movement_mechanism."4M1_engine_temperature_protection",VarCfg:="HMI_DB".IO_Tags.InCnf.DigIn_3_6);
           "DB_DigIn_I3.7"(ixVRaw:="4KT2", oxVal=>"HMI_DB".Crane_movement_mechanism."4M2_engine_temperature_protection",VarCfg:="HMI_DB".IO_Tags.InCnf.DigIn_3_7);
   END_REGION
   REGION A1_3
       "DB_DigIn_I4.0"(ixVRaw:="1BT1", oxVal=>"HMI_DB".Lifting_mechanism.Thermal_protection_braking_resistor,VarCfg:="HMI_DB".IO_Tags.InCnf.DigIn_4_0);
       "DB_DigIn_I4.1"(ixVRaw:="1K1", oxVal=>"HMI_DB".Lifting_mechanism.NSP_Upward_movement,VarCfg:="HMI_DB".IO_Tags.InCnf.DigIn_4_1);
       "DB_DigIn_I4.2"(ixVRaw:="1K2", oxVal=>"HMI_DB".Lifting_mechanism.NSP_Downward_movement,VarCfg:="HMI_DB".IO_Tags.InCnf.DigIn_4_2);
       "DB_DigIn_I4.3"(ixVRaw:="1K3", oxVal=>"HMI_DB".Lifting_mechanism.WP_Upward_movement,VarCfg:="HMI_DB".IO_Tags.InCnf.DigIn_4_3);
       "DB_DigIn_I4.4"(ixVRaw:="1K4", oxVal=>"HMI_DB".Lifting_mechanism.WP_Downward_movement,VarCfg:="HMI_DB".IO_Tags.InCnf.DigIn_4_4);
       "DB_DigIn_I4.5"(ixVRaw:="1K11", oxVal=>"HMI_DB".Lifting_mechanism."Exceeding_rated_load_115%",VarCfg:="HMI_DB".IO_Tags.InCnf.DigIn_4_5);
       "DB_DigIn_I4.6"(ixVRaw:="1K12", oxVal=>"HMI_DB".Lifting_mechanism.Loosening_ropes,VarCfg:="HMI_DB".IO_Tags.InCnf.DigIn_4_6);
       "DB_DigIn_I4.7"(ixVRaw:="1KT", oxVal=>"HMI_DB".Lifting_mechanism.Motor_temperature_protection,VarCfg:="HMI_DB".IO_Tags.InCnf.DigIn_4_7);
       "DB_DigIn_I5.0"(ixVRaw:="1K21", oxVal=>"HMI_DB".Lifting_mechanism."1YB1_Brake released",VarCfg:="HMI_DB".IO_Tags.InCnf.DigIn_5_0);
       "DB_DigIn_I5.1"(ixVRaw:="1K22", oxVal=>"HMI_DB".Lifting_mechanism."1YB1_Brake_applied",VarCfg:="HMI_DB".IO_Tags.InCnf.DigIn_5_1);
       "DB_DigIn_I5.2"(ixVRaw:="1K23", oxVal=>"HMI_DB".Lifting_mechanism."1YB1_Thickness_brake_pads_normal",VarCfg:="HMI_DB".IO_Tags.InCnf.DigIn_5_2);
       "DB_DigIn_I5.3"(ixVRaw:="1K31", oxVal=>"HMI_DB".Lifting_mechanism."1YB2_Brake released",VarCfg:="HMI_DB".IO_Tags.InCnf.DigIn_5_3);
       "DB_DigIn_I5.4"(ixVRaw:="1K32", oxVal=>"HMI_DB".Lifting_mechanism."1YB2_Brake_applied",VarCfg:="HMI_DB".IO_Tags.InCnf.DigIn_5_4);
       "DB_DigIn_I5.5"(ixVRaw:="1K33", oxVal=>"HMI_DB".Lifting_mechanism."1YB2_WP_MPP_disconnected_from_brake",VarCfg:="HMI_DB".IO_Tags.InCnf.DigIn_5_5);
       "DB_DigIn_I5.6"(ixVRaw:="1QF1", oxVal=>"HMI_DB".Lifting_mechanism."1YB1_Brake_rectifier_protection",VarCfg:="HMI_DB".IO_Tags.InCnf.DigIn_5_6);
       "DB_DigIn_I5.7"(ixVRaw:="1QF2", oxVal=>"HMI_DB".Lifting_mechanism."1YB2_Brake_rectifier_protection",VarCfg:="HMI_DB".IO_Tags.InCnf.DigIn_5_7);
       "DB_DigIn_I6.0"(ixVRaw:="3BT1", oxVal=>"HMI_DB".Trolley_movement_mechanism.Engine_temperature_protection,VarCfg:="HMI_DB".IO_Tags.InCnf.DigIn_6_0);
       "DB_DigIn_I6.1"(ixVRaw:="3K1", oxVal=>"HMI_DB".Trolley_movement_mechanism.NSP_Forward_movement,VarCfg:="HMI_DB".IO_Tags.InCnf.DigIn_6_1);
       "DB_DigIn_I6.2"(ixVRaw:="3K2", oxVal=>"HMI_DB".Trolley_movement_mechanism.WP_Forward_movement,VarCfg:="HMI_DB".IO_Tags.InCnf.DigIn_6_2);
       "DB_DigIn_I6.3"(ixVRaw:="3K3", oxVal=>"HMI_DB".Trolley_movement_mechanism.NSP_Backward_movement,VarCfg:="HMI_DB".IO_Tags.InCnf.DigIn_6_3);
       "DB_DigIn_I6.4"(ixVRaw:="3K4", oxVal=>"HMI_DB".Trolley_movement_mechanism.WP_Backward_movement,VarCfg:="HMI_DB".IO_Tags.InCnf.DigIn_6_4);
       "DB_DigIn_I6.5"(ixVRaw:="3K41", oxVal=>"HMI_DB".Trolley_movement_mechanism.MD_disconnected_from_drive,VarCfg:="HMI_DB".IO_Tags.InCnf.DigIn_6_5);
       "DB_DigIn_I6.6"(ixVRaw:="3KT", oxVal=>"HMI_DB".Trolley_movement_mechanism.Motor_temperature_protection,VarCfg:="HMI_DB".IO_Tags.InCnf.DigIn_6_6);
       "DB_DigIn_I6.7"(ixVRaw:="4K5", oxVal=>"HMI_DB".Crane_movement_mechanism.WP_Either_side_column,VarCfg:="HMI_DB".IO_Tags.InCnf.DigIn_6_7);
       "DB_DigIn_I7.0"(ixVRaw:="4BT1", oxVal=>"HMI_DB".Crane_movement_mechanism."4RT1_thermal_protection_braking_resistor",VarCfg:="HMI_DB".IO_Tags.InCnf.DigIn_7_0);
       "DB_DigIn_I7.1"(ixVRaw:="4BT2", oxVal=>"HMI_DB".Crane_movement_mechanism."4RT2_thermal_protection_braking_resistor",VarCfg:="HMI_DB".IO_Tags.InCnf.DigIn_7_1);
       "DB_DigIn_I7.2"(ixVRaw:="4K1", oxVal=>"HMI_DB".Crane_movement_mechanism.NSP_Left_movement,VarCfg:="HMI_DB".IO_Tags.InCnf.DigIn_7_2);
       "DB_DigIn_I7.3"(ixVRaw:="4K2", oxVal=>"HMI_DB".Crane_movement_mechanism.NSP_Right_movement,VarCfg:="HMI_DB".IO_Tags.InCnf.DigIn_7_3);
       "DB_DigIn_I7.4"(ixVRaw:="4K3", oxVal=>"HMI_DB".Crane_movement_mechanism.WP_Left_movement,VarCfg:="HMI_DB".IO_Tags.InCnf.DigIn_7_4);
       "DB_DigIn_I7.5"(ixVRaw:="4K4", oxVal=>"HMI_DB".Crane_movement_mechanism.WP_Right_movement,VarCfg:="HMI_DB".IO_Tags.InCnf.DigIn_7_5);
       "DB_DigIn_I7.6"(ixVRaw:="4K41", oxVal=>"HMI_DB".Crane_movement_mechanism."4SQ41_MD_disconnected_from_drive",VarCfg:="HMI_DB".IO_Tags.InCnf.DigIn_7_6);
       "DB_DigIn_I7.7"(ixVRaw:="4K42", oxVal=>"HMI_DB".Crane_movement_mechanism."4SQ42_MD_disconnected_from_drive",VarCfg:="HMI_DB".IO_Tags.InCnf.DigIn_7_7);
   END_REGION
   REGION A1_5
   "DB_AnIn_8"(iiVRaw:="1A1",orVal=>"HMI_DB".Lifting_mechanism.Torque_control,VarCfg:="HMI_DB".IO_Tags.InAnCfg.AnIn_0);
   "DB_AnIn_10"(VarCfg:="HMI_DB".IO_Tags.InAnCfg.AnIn_1);
   "DB_AnIn_12"(VarCfg:="HMI_DB".IO_Tags.InAnCfg.AnIn_2);
   "DB_AnIn_14"(VarCfg:="HMI_DB".IO_Tags.InAnCfg.AnIn_3);
   "DB_AnIn_16"(VarCfg:="HMI_DB".IO_Tags.InAnCfg.AnIn_4);
   "DB_AnIn_18"(VarCfg:="HMI_DB".IO_Tags.InAnCfg.AnIn_5);
   "DB_AnIn_20"(VarCfg:="HMI_DB".IO_Tags.InAnCfg.AnIn_6);
   "DB_AnIn_22"(VarCfg:="HMI_DB".IO_Tags.InAnCfg.AnIn_7);

   END_REGION

   END_REGION
END_FUNCTION

FUNCTION "FC_OutVar" : Void   // FC101, SCL
{ S7_Optimized_Access := 'TRUE' }
VERSION : 0.1
BEGIN
   REGION KZPTO
       REGION A1_5
           "DB_DigOut_Q0.0"(ixVRaw:="HMI_DB".Lifting_mechanism.CMD_Service_brake_On,oxVal=>"1KM1",VarCfg:="HMI_DB".IO_Tags.OutCfg.DigOut_0_0);
           "DB_DigOut_Q0.1"(ixVRaw:="HMI_DB".Lifting_mechanism."CMD_Built-in_brake_On",oxVal=>"1KM2",VarCfg:="HMI_DB".IO_Tags.OutCfg.DigOut_0_1);
           "DB_DigOut_Q0.2"(ixVRaw:="HMI_DB".Lifting_mechanism.CMD_Emergency_brake_On,oxVal=>"1KM3",VarCfg:="HMI_DB".IO_Tags.OutCfg.DigOut_0_2);
           "DB_DigOut_Q0.3"(ixVRaw:="HMI_DB".Trolley_movement_mechanism.CMD_Service_brake_On,oxVal=>"3KM1",VarCfg:="HMI_DB".IO_Tags.OutCfg.DigOut_0_3);
           "DB_DigOut_Q0.4"(ixVRaw:="HMI_DB".Crane_movement_mechanism.CMD_Service_brake_On,oxVal=>"4KM1",VarCfg:="HMI_DB".IO_Tags.OutCfg.DigOut_0_4);
           "DB_DigOut_Q0.5"(ixVRaw:="HMI_DB".PSM.CMD_Line_contactor_enable_permission,oxVal=>"6K1",VarCfg:="HMI_DB".IO_Tags.OutCfg.DigOut_0_5);
           "DB_DigOut_Q0.6"(ixVRaw:="HMI_DB".PSM.CMD_Line_contactor_Off,oxVal=>"6K2",VarCfg:="HMI_DB".IO_Tags.OutCfg.DigOut_0_6);
           "DB_DigOut_Q0.7"(ixVRaw:="HMI_DB".Sensors.CMD_Bell_On,oxVal=>"9K1",VarCfg:="HMI_DB".IO_Tags.OutCfg.DigOut_0_7);
           "DB_DigOut_Q1.0"(ixVRaw:="HMI_DB".Reserv.Q1_0,oxVal=>"Q1_0",VarCfg:="HMI_DB".IO_Tags.OutCfg.DigOut_1_0);
           "DB_DigOut_Q1.1"(ixVRaw:="HMI_DB".Reserv.Q1_1,oxVal=>"Q1_1",VarCfg:="HMI_DB".IO_Tags.OutCfg.DigOut_1_1);
           "DB_DigOut_Q1.2"(ixVRaw:="HMI_DB".Lifting_mechanism.HL_Drive_ready,oxVal=>"S1_1HL",VarCfg:="HMI_DB".IO_Tags.OutCfg.DigOut_1_2);
           "DB_DigOut_Q1.3"(ixVRaw:="HMI_DB".Trolley_movement_mechanism.HL_Drive_ready,oxVal=>"S1_3HL",VarCfg:="HMI_DB".IO_Tags.OutCfg.DigOut_1_3);
           "DB_DigOut_Q1.4"(ixVRaw:="HMI_DB".Crane_movement_mechanism.HL_Drive_ready,oxVal=>"S1_4HL",VarCfg:="HMI_DB".IO_Tags.OutCfg.DigOut_1_4);
           "DB_DigOut_Q1.5"(ixVRaw:="HMI_DB".PSM.HL_Line_contactor_On,oxVal=>"S1_6HL1",VarCfg:="HMI_DB".IO_Tags.OutCfg.DigOut_1_5);
           "DB_DigOut_Q1.6"(ixVRaw:="HMI_DB".PSM.HL_Input_voltage_abnormal,oxVal=>"S1_6HL2",VarCfg:="HMI_DB".IO_Tags.OutCfg.DigOut_1_6);
           "DB_DigOut_Q1.7"(ixVRaw:="HMI_DB".Reserv.Q1_7,oxVal=>"Q1_7",VarCfg:="HMI_DB".IO_Tags.OutCfg.DigOut_1_7);

       END_REGION
   END_REGION
END_FUNCTION

// folder: 2000_Tools

FUNCTION_BLOCK "FB_DigIn_16"   // FB2000, LAD
{ S7_Optimized_Access := 'TRUE' }
VERSION : 0.1
   VAR_INPUT
      Input_0 : Bool;
      Delay_Sec_0 : Real;
      Input_1 : Bool;
      Delay_Sec_1 : Real;
      Input_2 : Bool;
      Delay_Sec_2 : Real;
      Input_3 : Bool;
      Delay_Sec_3 : Real;
      Input_4 : Bool;
      Delay_Sec_4 : Real;
      Input_5 : Bool;
      Delay_Sec_5 : Real;
      Input_6 : Bool;
      Delay_Sec_6 : Real;
      Input_7 : Bool;
      Delay_Sec_7 : Real;
      Input_8 : Bool;
      Delay_Sec_8 : Real;
      Input_9 : Bool;
      Delay_Sec_9 : Real;
      Input_10 : Bool;
      Delay_Sec_10 : Real;
      Input_11 : Bool;
      Delay_Sec_11 : Real;
      Input_12 : Bool;
      Delay_Sec_12 : Real;
      Input_13 : Bool;
      Delay_Sec_13 : Real;
      Input_14 : Bool;
      Delay_Sec_14 : Real;
      Input_15 : Bool;
      Delay_Sec_15 : Real;
   END_VAR
   VAR_OUTPUT
      Alarm_0 : Bool;
      Alarm_1 : Bool;
      Alarm_2 : Bool;
      Alarm_3 : Bool;
      Alarm_4 : Bool;
      Alarm_5 : Bool;
      Alarm_6 : Bool;
      Alarm_7 : Bool;
      Alarm_8 : Bool;
      Alarm_9 : Bool;
      Alarm_10 : Bool;
      Alarm_11 : Bool;
      Alarm_12 : Bool;
      Alarm_13 : Bool;
      Alarm_14 : Bool;
      Alarm_15 : Bool;
      owHMI_Word : Word;
   END_VAR
   VAR
      Timer_0 : TON_TIME;
      Timer_1 : TON_TIME;
      Timer_2 : TON_TIME;
      Timer_3 : TON_TIME;
      Timer_4 : TON_TIME;
      Timer_5 : TON_TIME;
      Timer_6 : TON_TIME;
      Timer_7 : TON_TIME;
      Timer_8 : TON_TIME;
      Timer_9 : TON_TIME;
      Timer_10 : TON_TIME;
      Timer_11 : TON_TIME;
      Timer_12 : TON_TIME;
      Timer_13 : TON_TIME;
      Timer_14 : TON_TIME;
      Timer_15 : TON_TIME;
   END_VAR
   VAR_TEMP
      Tmp_Real : Real;
      Tmp_Time : DInt;
   END_VAR
BEGIN

REGION Network 1: Обработка аварии по входу №0 / Обробка аварії по входу №0
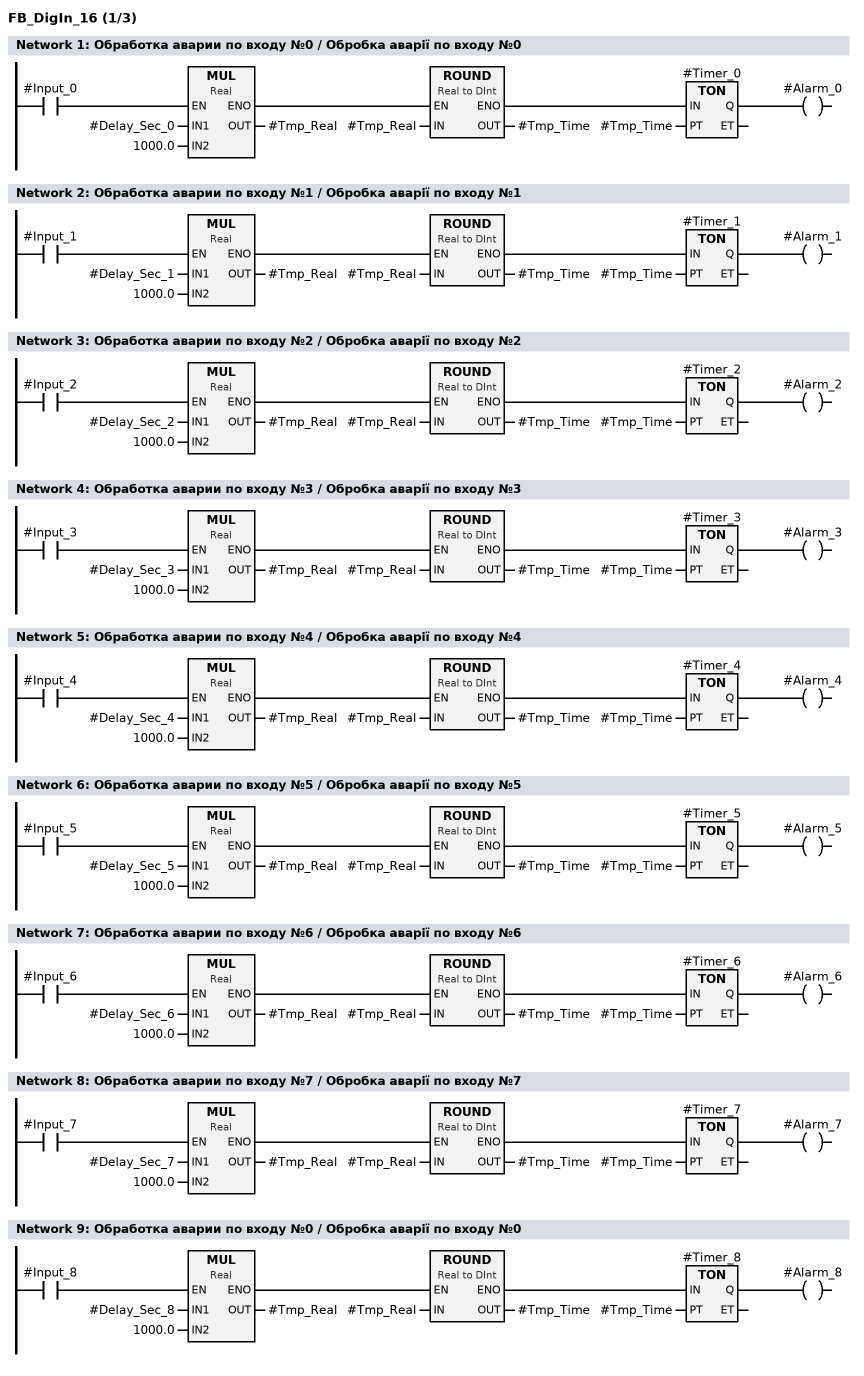
   IF #Input_0 THEN
       #Tmp_Real := #Delay_Sec_0 * 1000.0;
       #Tmp_Time := ROUND(#Tmp_Real);
   END_IF;
   #Timer_0(IN := #Input_0, PT := #Tmp_Time);   // TON
   #Alarm_0 := #Timer_0.Q;
END_REGION

REGION Network 2: Обработка аварии по входу №1 / Обробка аварії по входу №1
   IF #Input_1 THEN
       #Tmp_Real := #Delay_Sec_1 * 1000.0;
       #Tmp_Time := ROUND(#Tmp_Real);
   END_IF;
   #Timer_1(IN := #Input_1, PT := #Tmp_Time);   // TON
   #Alarm_1 := #Timer_1.Q;
END_REGION

REGION Network 3: Обработка аварии по входу №2 / Обробка аварії по входу №2
   IF #Input_2 THEN
       #Tmp_Real := #Delay_Sec_2 * 1000.0;
       #Tmp_Time := ROUND(#Tmp_Real);
   END_IF;
   #Timer_2(IN := #Input_2, PT := #Tmp_Time);   // TON
   #Alarm_2 := #Timer_2.Q;
END_REGION

REGION Network 4: Обработка аварии по входу №3 / Обробка аварії по входу №3
   IF #Input_3 THEN
       #Tmp_Real := #Delay_Sec_3 * 1000.0;
       #Tmp_Time := ROUND(#Tmp_Real);
   END_IF;
   #Timer_3(IN := #Input_3, PT := #Tmp_Time);   // TON
   #Alarm_3 := #Timer_3.Q;
END_REGION

REGION Network 5: Обработка аварии по входу №4 / Обробка аварії по входу №4
   IF #Input_4 THEN
       #Tmp_Real := #Delay_Sec_4 * 1000.0;
       #Tmp_Time := ROUND(#Tmp_Real);
   END_IF;
   #Timer_4(IN := #Input_4, PT := #Tmp_Time);   // TON
   #Alarm_4 := #Timer_4.Q;
END_REGION

REGION Network 6: Обработка аварии по входу №5 / Обробка аварії по входу №5
   IF #Input_5 THEN
       #Tmp_Real := #Delay_Sec_5 * 1000.0;
       #Tmp_Time := ROUND(#Tmp_Real);
   END_IF;
   #Timer_5(IN := #Input_5, PT := #Tmp_Time);   // TON
   #Alarm_5 := #Timer_5.Q;
END_REGION

REGION Network 7: Обработка аварии по входу №6 / Обробка аварії по входу №6
   IF #Input_6 THEN
       #Tmp_Real := #Delay_Sec_6 * 1000.0;
       #Tmp_Time := ROUND(#Tmp_Real);
   END_IF;
   #Timer_6(IN := #Input_6, PT := #Tmp_Time);   // TON
   #Alarm_6 := #Timer_6.Q;
END_REGION

REGION Network 8: Обработка аварии по входу №7 / Обробка аварії по входу №7
   IF #Input_7 THEN
       #Tmp_Real := #Delay_Sec_7 * 1000.0;
       #Tmp_Time := ROUND(#Tmp_Real);
   END_IF;
   #Timer_7(IN := #Input_7, PT := #Tmp_Time);   // TON
   #Alarm_7 := #Timer_7.Q;
END_REGION

REGION Network 9: Обработка аварии по входу №0 / Обробка аварії по входу №0
   IF #Input_8 THEN
       #Tmp_Real := #Delay_Sec_8 * 1000.0;
       #Tmp_Time := ROUND(#Tmp_Real);
   END_IF;
   #Timer_8(IN := #Input_8, PT := #Tmp_Time);   // TON
   #Alarm_8 := #Timer_8.Q;
END_REGION

REGION Network 10: Обработка аварии по входу №0 / Обробка аварії по входу №0
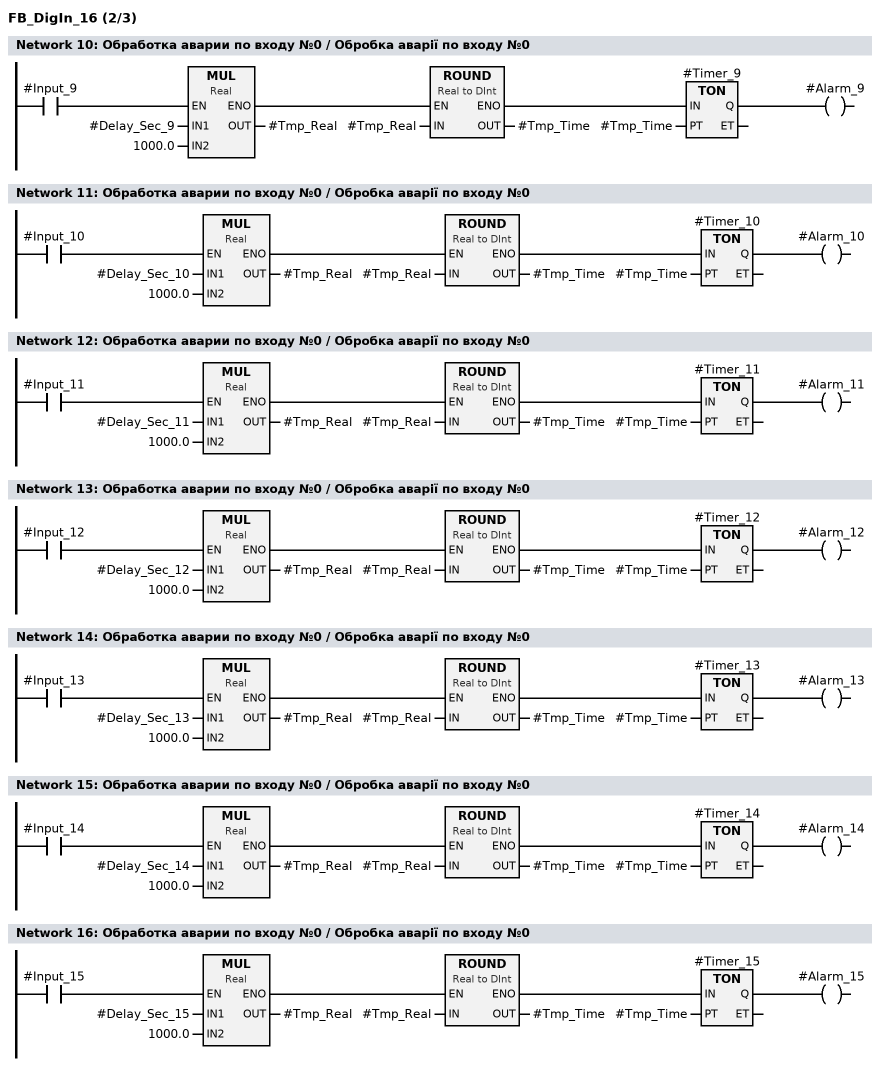
   IF #Input_9 THEN
       #Tmp_Real := #Delay_Sec_9 * 1000.0;
       #Tmp_Time := ROUND(#Tmp_Real);
   END_IF;
   #Timer_9(IN := #Input_9, PT := #Tmp_Time);   // TON
   #Alarm_9 := #Timer_9.Q;
END_REGION

REGION Network 11: Обработка аварии по входу №0 / Обробка аварії по входу №0
   IF #Input_10 THEN
       #Tmp_Real := #Delay_Sec_10 * 1000.0;
       #Tmp_Time := ROUND(#Tmp_Real);
   END_IF;
   #Timer_10(IN := #Input_10, PT := #Tmp_Time);   // TON
   #Alarm_10 := #Timer_10.Q;
END_REGION

REGION Network 12: Обработка аварии по входу №0 / Обробка аварії по входу №0
   IF #Input_11 THEN
       #Tmp_Real := #Delay_Sec_11 * 1000.0;
       #Tmp_Time := ROUND(#Tmp_Real);
   END_IF;
   #Timer_11(IN := #Input_11, PT := #Tmp_Time);   // TON
   #Alarm_11 := #Timer_11.Q;
END_REGION

REGION Network 13: Обработка аварии по входу №0 / Обробка аварії по входу №0
   IF #Input_12 THEN
       #Tmp_Real := #Delay_Sec_12 * 1000.0;
       #Tmp_Time := ROUND(#Tmp_Real);
   END_IF;
   #Timer_12(IN := #Input_12, PT := #Tmp_Time);   // TON
   #Alarm_12 := #Timer_12.Q;
END_REGION

REGION Network 14: Обработка аварии по входу №0 / Обробка аварії по входу №0
   IF #Input_13 THEN
       #Tmp_Real := #Delay_Sec_13 * 1000.0;
       #Tmp_Time := ROUND(#Tmp_Real);
   END_IF;
   #Timer_13(IN := #Input_13, PT := #Tmp_Time);   // TON
   #Alarm_13 := #Timer_13.Q;
END_REGION

REGION Network 15: Обработка аварии по входу №0 / Обробка аварії по входу №0
   IF #Input_14 THEN
       #Tmp_Real := #Delay_Sec_14 * 1000.0;
       #Tmp_Time := ROUND(#Tmp_Real);
   END_IF;
   #Timer_14(IN := #Input_14, PT := #Tmp_Time);   // TON
   #Alarm_14 := #Timer_14.Q;
END_REGION

REGION Network 16: Обработка аварии по входу №0 / Обробка аварії по входу №0
   IF #Input_15 THEN
       #Tmp_Real := #Delay_Sec_15 * 1000.0;
       #Tmp_Time := ROUND(#Tmp_Real);
   END_IF;
   #Timer_15(IN := #Input_15, PT := #Tmp_Time);   // TON
   #Alarm_15 := #Timer_15.Q;
END_REGION

REGION Network 17: Формування статусних слів
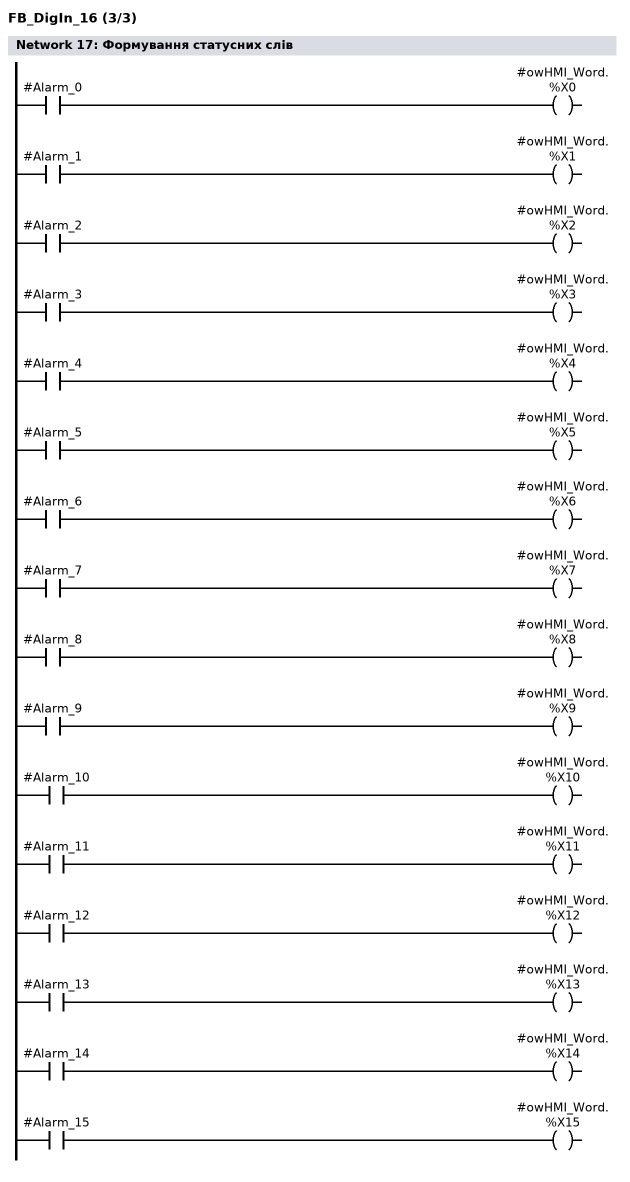
   RUNG wire#powerrail
      Contact( #Alarm_0 )
      Coil( #owHMI_Word.%X0 )
   END_RUNG
   RUNG wire#powerrail
      Contact( #Alarm_1 )
      Coil( #owHMI_Word.%X1 )
   END_RUNG
   RUNG wire#powerrail
      Contact( #Alarm_2 )
      Coil( #owHMI_Word.%X2 )
   END_RUNG
   RUNG wire#powerrail
      Contact( #Alarm_3 )
      Coil( #owHMI_Word.%X3 )
   END_RUNG
   RUNG wire#powerrail
      Contact( #Alarm_4 )
      Coil( #owHMI_Word.%X4 )
   END_RUNG
   RUNG wire#powerrail
      Contact( #Alarm_5 )
      Coil( #owHMI_Word.%X5 )
   END_RUNG
   RUNG wire#powerrail
      Contact( #Alarm_6 )
      Coil( #owHMI_Word.%X6 )
   END_RUNG
   RUNG wire#powerrail
      Contact( #Alarm_7 )
      Coil( #owHMI_Word.%X7 )
   END_RUNG
   RUNG wire#powerrail
      Contact( #Alarm_8 )
      Coil( #owHMI_Word.%X8 )
   END_RUNG
   RUNG wire#powerrail
      Contact( #Alarm_9 )
      Coil( #owHMI_Word.%X9 )
   END_RUNG
   RUNG wire#powerrail
      Contact( #Alarm_10 )
      Coil( #owHMI_Word.%X10 )
   END_RUNG
   RUNG wire#powerrail
      Contact( #Alarm_11 )
      Coil( #owHMI_Word.%X11 )
   END_RUNG
   RUNG wire#powerrail
      Contact( #Alarm_12 )
      Coil( #owHMI_Word.%X12 )
   END_RUNG
   RUNG wire#powerrail
      Contact( #Alarm_13 )
      Coil( #owHMI_Word.%X13 )
   END_RUNG
   RUNG wire#powerrail
      Contact( #Alarm_14 )
      Coil( #owHMI_Word.%X14 )
   END_RUNG
   RUNG wire#powerrail
      Contact( #Alarm_15 )
      Coil( #owHMI_Word.%X15 )
   END_RUNG
   // the same network as SCL:
   #owHMI_Word.%X0 := #Alarm_0;
   #owHMI_Word.%X1 := #Alarm_1;
   #owHMI_Word.%X2 := #Alarm_2;
   #owHMI_Word.%X3 := #Alarm_3;
   #owHMI_Word.%X4 := #Alarm_4;
   #owHMI_Word.%X5 := #Alarm_5;
   #owHMI_Word.%X6 := #Alarm_6;
   #owHMI_Word.%X7 := #Alarm_7;
   #owHMI_Word.%X8 := #Alarm_8;
   #owHMI_Word.%X9 := #Alarm_9;
   #owHMI_Word.%X10 := #Alarm_10;
   #owHMI_Word.%X11 := #Alarm_11;
   #owHMI_Word.%X12 := #Alarm_12;
   #owHMI_Word.%X13 := #Alarm_13;
   #owHMI_Word.%X14 := #Alarm_14;
   #owHMI_Word.%X15 := #Alarm_15;
END_REGION
END_FUNCTION_BLOCK

FUNCTION_BLOCK "FB_DigIn_16_XOR"   // FB2001, LAD
{ S7_Optimized_Access := 'TRUE' }
VERSION : 0.1
   VAR_INPUT
      Input_0 : Bool;
      Delay_Sec_0 : Real;
      Input_1 : Bool;
      Delay_Sec_1 : Real;
      Input_2 : Bool;
      Delay_Sec_2 : Real;
      Input_3 : Bool;
      Delay_Sec_3 : Real;
      Input_4 : Bool;
      Delay_Sec_4 : Real;
      Input_5 : Bool;
      Delay_Sec_5 : Real;
      Input_6 : Bool;
      Delay_Sec_6 : Real;
      Input_7 : Bool;
      Delay_Sec_7 : Real;
      Input_8 : Bool;
      Delay_Sec_8 : Real;
      Input_9 : Bool;
      Delay_Sec_9 : Real;
      Input_10 : Bool;
      Delay_Sec_10 : Real;
      Input_11 : Bool;
      Delay_Sec_11 : Real;
      Input_12 : Bool;
      Delay_Sec_12 : Real;
      Input_13 : Bool;
      Delay_Sec_13 : Real;
      Input_14 : Bool;
      Delay_Sec_14 : Real;
      Input_15 : Bool;
      Delay_Sec_15 : Real;
      ixInit : Bool;   // Ініціалізація
   END_VAR
   VAR_OUTPUT
      Alarm_0 : Bool;
      Alarm_1 : Bool;
      Alarm_2 : Bool;
      Alarm_3 : Bool;
      Alarm_4 : Bool;
      Alarm_5 : Bool;
      Alarm_6 : Bool;
      Alarm_7 : Bool;
      Alarm_8 : Bool;
      Alarm_9 : Bool;
      Alarm_10 : Bool;
      Alarm_11 : Bool;
      Alarm_12 : Bool;
      Alarm_13 : Bool;
      Alarm_14 : Bool;
      Alarm_15 : Bool;
      owHMI_Word : Word;
   END_VAR
   VAR
      Timer_0 : TON_TIME;
      Timer_1 : TON_TIME;
      Timer_2 : TON_TIME;
      Timer_3 : TON_TIME;
      Timer_4 : TON_TIME;
      Timer_5 : TON_TIME;
      Timer_6 : TON_TIME;
      Timer_7 : TON_TIME;
      Timer_8 : TON_TIME;
      Timer_9 : TON_TIME;
      Timer_10 : TON_TIME;
      Timer_11 : TON_TIME;
      Timer_12 : TON_TIME;
      Timer_13 : TON_TIME;
      Timer_14 : TON_TIME;
      Timer_15 : TON_TIME;
      sarxArrayFlanke : Array[0..15] of Bool;   // Help Array for flanke
      sarxArrayMerkers : Array[0..15] of Bool;   // Help Array for merkers
   END_VAR
   VAR_TEMP
      Tmp_Real : Real;
      Tmp_Time : DInt;
   END_VAR
   VAR_TEMP   // added for the SCL form of the ladder/FBD networks
      _w1 : Bool;
   END_VAR
BEGIN

REGION Network 1: Умови стрибка
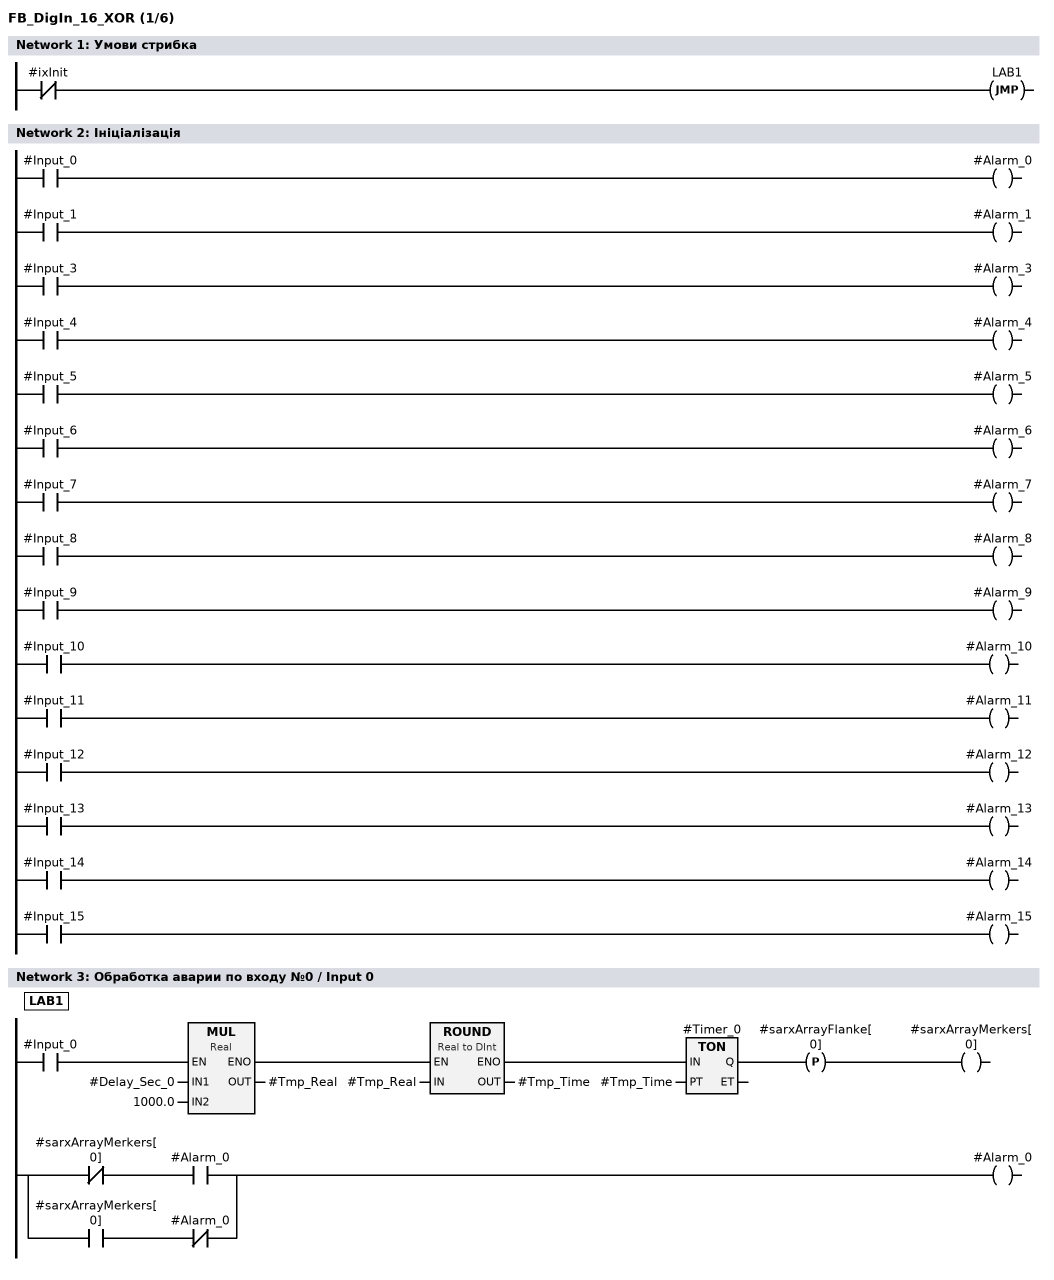
   RUNG wire#powerrail
      I_Contact( #ixInit )
      JumpCoil( LAB1 )
   END_RUNG
   // the same network as SCL:
   IF NOT #ixInit THEN GOTO LAB1; END_IF;
END_REGION

REGION Network 2: Ініціалізація
   RUNG wire#powerrail
      Contact( #Input_0 )
      Coil( #Alarm_0 )
   END_RUNG
   RUNG wire#powerrail
      Contact( #Input_1 )
      Coil( #Alarm_1 )
   END_RUNG
   RUNG wire#powerrail
      Contact( #Input_3 )
      Coil( #Alarm_3 )
   END_RUNG
   RUNG wire#powerrail
      Contact( #Input_4 )
      Coil( #Alarm_4 )
   END_RUNG
   RUNG wire#powerrail
      Contact( #Input_5 )
      Coil( #Alarm_5 )
   END_RUNG
   RUNG wire#powerrail
      Contact( #Input_6 )
      Coil( #Alarm_6 )
   END_RUNG
   RUNG wire#powerrail
      Contact( #Input_7 )
      Coil( #Alarm_7 )
   END_RUNG
   RUNG wire#powerrail
      Contact( #Input_8 )
      Coil( #Alarm_8 )
   END_RUNG
   RUNG wire#powerrail
      Contact( #Input_9 )
      Coil( #Alarm_9 )
   END_RUNG
   RUNG wire#powerrail
      Contact( #Input_10 )
      Coil( #Alarm_10 )
   END_RUNG
   RUNG wire#powerrail
      Contact( #Input_11 )
      Coil( #Alarm_11 )
   END_RUNG
   RUNG wire#powerrail
      Contact( #Input_12 )
      Coil( #Alarm_12 )
   END_RUNG
   RUNG wire#powerrail
      Contact( #Input_13 )
      Coil( #Alarm_13 )
   END_RUNG
   RUNG wire#powerrail
      Contact( #Input_14 )
      Coil( #Alarm_14 )
   END_RUNG
   RUNG wire#powerrail
      Contact( #Input_15 )
      Coil( #Alarm_15 )
   END_RUNG
   // the same network as SCL:
   #Alarm_0 := #Input_0;
   #Alarm_1 := #Input_1;
   #Alarm_3 := #Input_3;
   #Alarm_4 := #Input_4;
   #Alarm_5 := #Input_5;
   #Alarm_6 := #Input_6;
   #Alarm_7 := #Input_7;
   #Alarm_8 := #Input_8;
   #Alarm_9 := #Input_9;
   #Alarm_10 := #Input_10;
   #Alarm_11 := #Input_11;
   #Alarm_12 := #Input_12;
   #Alarm_13 := #Input_13;
   #Alarm_14 := #Input_14;
   #Alarm_15 := #Input_15;
END_REGION

